BEGIN
   MachineConfig[0]."Unit Sep"."EM - 100"."L-GREEN".CW.ENABLE := True;
   MachineConfig[0]."Unit Sep"."EM - 100"."L-GREEN".CW.EXIST := False;
   MachineConfig[1].Machine."Family" := 1;
   MachineConfig[1].Machine.TypeNo := 1;
   MachineConfig[1].Machine.Range := 2;
   MachineConfig[1].Machine.SepType := 1;
   MachineConfig[1].Machine.Frame := 4;
   MachineConfig[1].Machine.DchSystem := 1;
   MachineConfig[1].Machine.Spare_1 := 1;
   MachineConfig[1].Machine.FeedPump := 1;
   MachineConfig[1].Machine.InlineCarbonation := 1;
   MachineConfig[1].Machine.eWON := 1;
   MachineConfig[1]."Unit Sep"."EM - 100"."L-GREEN".CW.ENABLE := true;
   MachineConfig[1]."Unit Sep"."EM - 100"."L-YELLOW".Tag := 'L-BLUE';
   MachineConfig[1]."Unit Sep"."EM - 100"."L-RED".CW.EXIST := True;
   MachineConfig[1]."Unit Sep"."EM - 100".EMS.CW.EXIST := True;
   MachineConfig[1]."Unit Sep"."EM - 100".EMS.Address := 180;
   MachineConfig[1]."Unit Sep"."EM - 100".UPS.CW.ENABLE := False;
   MachineConfig[1]."Unit Sep"."EM - 100".UPS.CW.EXIST := False;
   MachineConfig[1]."Unit Sep"."EM - 100".UPS.Address := 181;
   MachineConfig[1]."Unit Sep"."EM - 100".EWON.CW.ENABLE := True;
   MachineConfig[1]."Unit Sep"."EM - 100".EWON.CW.EXIST := True;
   MachineConfig[1]."Unit Sep"."EM - 100"."LT BUF".CW.ENABLE := False;
   MachineConfig[1]."Unit Sep"."EM - 400"."AV409-1".CW.ENABLE := False;
   MachineConfig[1]."Unit Sep"."EM - 400"."FCV409-1".CW.ENABLE := False;
   MachineConfig[1]."Unit Sep"."EM - 400"."FIS409-1".CW.ENABLE := false;
   MachineConfig[1]."Unit Sep"."EM - 400"."FIT409-1".CW.ENABLE := False;
   MachineConfig[1]."Unit Sep"."EM - 600"."AV615-1".ACT_OUT_ADD := 173;
   MachineConfig[1]."Unit Sep"."EM - 600"."AV63X/441-1".TAG := 'AV635-1';
   MachineConfig[1]."Unit Sep"."EM - 600"."AV63X/441-1".CW.ENABLE := True;
   MachineConfig[1]."Unit Sep"."EM - 600"."AV63X/441-1".ACT_OUT_ADD := 174;
   MachineConfig[1]."Unit Sep"."EM - 600"."FIS615-1".CW.ENABLE := false;
   MachineConfig[1]."Unit Sep"."EM - 600"."FIS635-1".CW.ENABLE := true;
   MachineConfig[1]."Unit Sep"."EM - 600"."FIS635-1".CW.EXIST := True;
   MachineConfig[1]."Unit Sep"."EM - 701".M701."TYPE" := 2;
   MachineConfig[1]."Unit Sep"."EM - 701".M701.FB_RUN_ADD := 8;
   MachineConfig[1]."Unit Sep"."EM - 701".M701.FB_RDY_ADD := 8;
   MachineConfig[1]."Unit Sep"."EM - 701".M701.OUT_ACT_ADD := 512;
   MachineConfig[1]."Unit Sep"."EM - 701".M701.OUT_RST_ADD := 8;
   MachineConfig[1]."Unit Sep"."EM - 701".M701_AMPS.CW.EXIST := True;
   MachineConfig[1]."Unit Sep"."EM - 730".TS730.CW.ENABLE := true;
   MachineConfig[1]."Unit Sep"."EM - 730".TS730.CW.EXIST := True;
   MachineConfig[1]."Unit Sep"."EM - 730".TS730.Address := 184;
   MachineConfig[1]."Unit Sep"."EM - 740"."P+F PS".Address := 180;
   MachineConfig[1]."Unit Sep"."EM - 740"."P+F OS".CW.EXIST := True;
   MachineConfig[1]."Unit Sep"."EM - 740"."P+F OS".Address := 182;
   MachineConfig[1]."Unit Sep"."EM - 740"."P+F ERROR".Address := 183;
   MachineConfig[1]."Unit Sep"."EM - 750".YT75X.CW.ENABLE := False;
   MachineConfig[1]."Unit Process"."EM - 201"."AV201-1".CW.ENABLE := true;
   MachineConfig[1]."Unit Process"."EM - 201"."AV201-1".CW.FB_CLS_EN := false;
   MachineConfig[1]."Unit Process"."EM - 201"."AV201-1".CW.FB_OPN_EN := false;
   MachineConfig[1]."Unit Process"."EM - 201"."AV201-1".CW.VLV_W_FB := false;
   MachineConfig[1]."Unit Process"."EM - 201"."AV201-1".FB_OPN_ADD := 8;
   MachineConfig[1]."Unit Process"."EM - 201"."AV201-1".FB_CLS_ADD := 8;
   MachineConfig[1]."Unit Process"."EM - 201"."AV201-1".ACT_OUT_ADD := 160;
   MachineConfig[1]."Unit Process"."EM - 201"."FCV201-1".CW.ENABLE := False;
   MachineConfig[1]."Unit Process"."EM - 201"."FIT201-1".CW.ENABLE := True;
   MachineConfig[1]."Unit Process"."EM - 201"."FIT201-1".CW.EXIST := True;
   MachineConfig[1]."Unit Process"."EM - 201"."FIT201-1"."Type" := 0;
   MachineConfig[1]."Unit Process"."EM - 201"."FIT201-1".Address := 88;
   MachineConfig[1]."Unit Process"."EM - 201"."FIT201-1".Max := 10000.0;
   MachineConfig[1]."Unit Process"."EM - 201"."LA201-1".CW.ENABLE := False;
   MachineConfig[1]."Unit Process"."EM - 201"."PIT201-1".CW.ENABLE := False;
   MachineConfig[1]."Unit Process"."EM - 22X"."FIT22X-1".CW.ENABLE := False;
   MachineConfig[1]."Unit Process"."EM - 22X"."PIT22X-1".CW.ENABLE := False;
   MachineConfig[1]."Unit Process"."EM - 22X"."QT220-1".CW.ENABLE := True;
   MachineConfig[1]."Unit Process"."EM - 22X"."QT220-1".CW.EXIST := False;
   MachineConfig[1]."Unit Process"."EM - 22X"."PCV22X-1".CW.ENABLE := False;
   MachineConfig[1]."Unit Process"."EM - 340"."AV340-1".CW.ENABLE := False;
   MachineConfig[1]."Unit Process"."EM - 340"."PIS340-1".Tag := 'PS301-1';
   MachineConfig[1]."Unit Process"."EM - 340"."PIS340-1".CW.INPUT := False;
   MachineConfig[1]."Unit Dch"."EM - 222"."LS222-1".CW.ENABLE := False;
   MachineConfig[1]."Unit Dch"."EM - 222"."P222-1".CW.EXIST := False;
   MachineConfig[1]."Unit Dch"."EM - 222"."P222-1".FB_RUN_ADD := 194;
   MachineConfig[1]."Unit Dch"."EM - 222"."P222-1".FB_RDY_ADD := 195;
   MachineConfig[1]."Unit Dch"."EM - 222"."P222-1".OUT_ACT_ADD := 182;
   MachineConfig[1]."Unit Dch"."EM - 222"."TS222-1".CW.ENABLE := False;
   MachineConfig[1]."Unit Dch"."EM - 222"."TT222-1".CW.ENABLE := False;
   MachineConfig[1]."Unit Dch"."EM - 300"."AV301-1".CW.ENABLE := True;
   MachineConfig[1]."Unit Dch"."EM - 300"."AV301-1".CW.FB_CLS_EN := false;
   MachineConfig[1]."Unit Dch"."EM - 300"."AV301-1".CW.FB_OPN_EN := false;
   MachineConfig[1]."Unit Dch"."EM - 300"."AV301-1".CW.VLV_W_FB := false;
   MachineConfig[1]."Unit Dch"."EM - 300"."AV301-1".FB_OPN_ADD := 8;
   MachineConfig[1]."Unit Dch"."EM - 300"."AV301-1".FB_CLS_ADD := 8;
   MachineConfig[1]."Unit Dch"."EM - 300"."AV301-1".ACT_OUT_ADD := 163;
   MachineConfig[1]."Unit Dch"."EM - 300"."AV304-1".ACT_OUT_ADD := 163;
   MachineConfig[1]."Unit Dch"."EM - 300"."AV320-1".CW.ENABLE := true;
   MachineConfig[1]."Unit Dch"."EM - 300"."AV320-1".CW.FB_CLS_EN := false;
   MachineConfig[1]."Unit Dch"."EM - 300"."AV320-1".CW.FB_OPN_EN := false;
   MachineConfig[1]."Unit Dch"."EM - 300"."AV320-1".CW.VLV_W_FB := false;
   MachineConfig[1]."Unit Dch"."EM - 300"."AV320-1".FB_OPN_ADD := 8;
   MachineConfig[1]."Unit Dch"."EM - 300"."AV320-1".FB_CLS_ADD := 8;
   MachineConfig[1]."Unit Dch"."EM - 300"."AV320-1".ACT_OUT_ADD := 164;
   MachineConfig[1]."Unit Dch"."EM - 300"."PS301-1".CW.ENABLE := True;
   MachineConfig[1]."Unit Dch"."EM - 300"."PS301-1".CW.EXIST := True;
   MachineConfig[1]."Unit Dch"."EM - 375"."AV37X-1".TAG := 'AV376-1';
   MachineConfig[1]."Unit Dch"."EM - 375"."AV37X-1".CW.ENABLE := true;
   MachineConfig[1]."Unit Dch"."EM - 375"."AV37X-1".ACT_OUT_ADD := 166;
   MachineConfig[1]."Unit Dch"."EM - 375".LS793.CW.ENABLE := True;
   MachineConfig[1]."Unit Dch"."EM - 375".LS793.CW.EXIST := True;
   MachineConfig[1]."Unit Dch"."EM - 375"."PIS375-1".CW.ENABLE := false;
   MachineConfig[1]."Unit Dch"."EM - 506".IP506a.CW.ENABLE := False;
   MachineConfig[1]."Unit Dch"."EM - 506".AVDCH.TAG := 'AV372-1';
   MachineConfig[1]."Unit Dch"."EM - 506".AVDCH.CW.ENABLE := True;
   MachineConfig[1]."Unit Dch"."EM - 506".AVDCH.ACT_OUT_ADD := 167;
   MachineConfig[1].Options."EM - P201"."P201-1".FB_RUN_ADD := 196;
   MachineConfig[1].Options."EM - P201"."P201-1".FB_RDY_ADD := 197;
   MachineConfig[1].Options."EM - P201"."P201-1".OUT_ACT_ADD := 183;
   MachineConfig[1].Options."EM - P201"."P201-1".OUT_RST_ADD := 184;
   MachineConfig[2].Machine."Family" := 1;
   MachineConfig[2].Machine.TypeNo := 2;
   MachineConfig[2].Machine.Range := 2;
   MachineConfig[2].Machine.SepType := 1;
   MachineConfig[2].Machine.Frame := 3;
   MachineConfig[2].Machine.DchSystem := 1;
   MachineConfig[2].Machine.Spare_1 := 1;
   MachineConfig[2].Machine.FeedPump := 1;
   MachineConfig[2].Machine.InlineCarbonation := 1;
   MachineConfig[2].Machine.eWON := 1;
   MachineConfig[2].Machine.ALBufferTank := 1;
   MachineConfig[2]."Unit Sep"."EM - 100"."L-GREEN".CW.ENABLE := true;
   MachineConfig[2]."Unit Sep"."EM - 100"."L-YELLOW".Tag := 'L-BLUE';
   MachineConfig[2]."Unit Sep"."EM - 100".EMS.Address := 180;
   MachineConfig[2]."Unit Sep"."EM - 100".UPS.CW.ENABLE := False;
   MachineConfig[2]."Unit Sep"."EM - 100".UPS.Address := 181;
   MachineConfig[2]."Unit Sep"."EM - 100".EWON.CW.ENABLE := True;
   MachineConfig[2]."Unit Sep"."EM - 100".EWON.CW.EXIST := True;
   MachineConfig[2]."Unit Sep"."EM - 400"."AV409-1".CW.ENABLE := False;
   MachineConfig[2]."Unit Sep"."EM - 400"."FCV409-1".CW.ENABLE := False;
   MachineConfig[2]."Unit Sep"."EM - 400"."FIS409-1".CW.ENABLE := false;
   MachineConfig[2]."Unit Sep"."EM - 400"."FIT409-1".CW.ENABLE := False;
   MachineConfig[2]."Unit Sep"."EM - 600"."AV63X/441-1".TAG := 'AV635-1';
   MachineConfig[2]."Unit Sep"."EM - 600"."AV63X/441-1".CW.ENABLE := True;
   MachineConfig[2]."Unit Sep"."EM - 600"."AV63X/441-1".ACT_OUT_ADD := 174;
   MachineConfig[2]."Unit Sep"."EM - 600"."FIS615-1".CW.ENABLE := False;
   MachineConfig[2]."Unit Sep"."EM - 600"."FIS635-1".CW.ENABLE := True;
   MachineConfig[2]."Unit Sep"."EM - 600"."FIS635-1".CW.EXIST := True;
   MachineConfig[2]."Unit Sep"."EM - 701".M701."TYPE" := 2;
   MachineConfig[2]."Unit Sep"."EM - 701".M701.FB_RUN_ADD := 8;
   MachineConfig[2]."Unit Sep"."EM - 701".M701.FB_RDY_ADD := 8;
   MachineConfig[2]."Unit Sep"."EM - 701".M701.OUT_ACT_ADD := 512;
   MachineConfig[2]."Unit Sep"."EM - 701".M701.OUT_RST_ADD := 8;
   MachineConfig[2]."Unit Sep"."EM - 730".TS730.CW.ENABLE := true;
   MachineConfig[2]."Unit Sep"."EM - 730".TS730.Address := 184;
   MachineConfig[2]."Unit Sep"."EM - 740"."P+F PS".Address := 180;
   MachineConfig[2]."Unit Sep"."EM - 740"."P+F OS".Address := 182;
   MachineConfig[2]."Unit Sep"."EM - 740"."P+F ERROR".Address := 183;
   MachineConfig[2]."Unit Sep"."EM - 750".YT75X.Tag := 'YT752';
   MachineConfig[2]."Unit Sep"."EM - 750".YT75X.CW.ENABLE := True;
   MachineConfig[2]."Unit Sep"."EM - 750".YT75X.Address := 78;
   MachineConfig[2]."Unit Sep"."EM - 750".YT75X.Min := 2.3;
   MachineConfig[2]."Unit Sep"."EM - 750".YT75X.Max := 5.5;
   MachineConfig[2]."Unit Sep"."EM - 750".YT75X.EU := 51;
   MachineConfig[2]."Unit Process"."EM - 201"."AV201-1".CW.ENABLE := True;
   MachineConfig[2]."Unit Process"."EM - 201"."AV201-1".CW.FB_CLS_EN := false;
   MachineConfig[2]."Unit Process"."EM - 201"."AV201-1".CW.FB_OPN_EN := false;
   MachineConfig[2]."Unit Process"."EM - 201"."AV201-1".CW.VLV_W_FB := false;
   MachineConfig[2]."Unit Process"."EM - 201"."AV201-1".FB_OPN_ADD := 8;
   MachineConfig[2]."Unit Process"."EM - 201"."AV201-1".FB_CLS_ADD := 8;
   MachineConfig[2]."Unit Process"."EM - 201"."AV201-1".ACT_OUT_ADD := 160;
   MachineConfig[2]."Unit Process"."EM - 201"."FCV201-1".CW.EXIST := false;
   MachineConfig[2]."Unit Process"."EM - 201"."FIT201-1"."Type" := 0;
   MachineConfig[2]."Unit Process"."EM - 201"."FIT201-1".Address := 88;
   MachineConfig[2]."Unit Process"."EM - 201"."FIT201-1".Max := 10000.0;
   MachineConfig[2]."Unit Process"."EM - 201"."LA201-1".CW.ENABLE := False;
   MachineConfig[2]."Unit Process"."EM - 201"."PIT201-1".CW.ENABLE := true;
   MachineConfig[2]."Unit Process"."EM - 201"."PIT201-1".CW.EXIST := false;
   MachineConfig[2]."Unit Process"."EM - 201"."QT201-1".CW.ENABLE := True;
   MachineConfig[2]."Unit Process"."EM - 22X"."AV220-1".CW.FB_CLS_EN := false;
   MachineConfig[2]."Unit Process"."EM - 22X"."AV220-1".CW.FB_OPN_EN := false;
   MachineConfig[2]."Unit Process"."EM - 22X"."AV220-1".CW.VLV_W_FB := false;
   MachineConfig[2]."Unit Process"."EM - 22X"."AV220-1".FB_OPN_ADD := 8;
   MachineConfig[2]."Unit Process"."EM - 22X"."AV220-1".FB_CLS_ADD := 8;
   MachineConfig[2]."Unit Process"."EM - 22X"."AV220-1".ACT_OUT_ADD := 162;
   MachineConfig[2]."Unit Process"."EM - 22X"."FIT22X-1".CW.ENABLE := false;
   MachineConfig[2]."Unit Process"."EM - 22X"."PIT22X-1".CW.EXIST := False;
   MachineConfig[2]."Unit Process"."EM - 22X"."QT220-1".CW.ENABLE := True;
   MachineConfig[2]."Unit Process"."EM - 22X"."QT220-1".CW.EXIST := False;
   MachineConfig[2]."Unit Process"."EM - 22X"."PCV22X-1".CW.ENABLE := False;
   MachineConfig[2]."Unit Process"."EM - 340"."AV340-1".CW.ENABLE := false;
   MachineConfig[2]."Unit Process"."EM - 340"."AV340-1".CW.FB_CLS_EN := false;
   MachineConfig[2]."Unit Process"."EM - 340"."AV340-1".CW.FB_OPN_EN := false;
   MachineConfig[2]."Unit Process"."EM - 340"."AV340-1".CW.EXIST := false;
   MachineConfig[2]."Unit Process"."EM - 340"."AV340-1".CW.VLV_W_FB := false;
   MachineConfig[2]."Unit Process"."EM - 340"."AV340-1".FB_OPN_ADD := 8;
   MachineConfig[2]."Unit Process"."EM - 340"."AV340-1".FB_CLS_ADD := 8;
   MachineConfig[2]."Unit Process"."EM - 340"."AV340-1".ACT_OUT_ADD := 8;
   MachineConfig[2]."Unit Dch"."EM - 222"."LS222-1".CW.ENABLE := False;
   MachineConfig[2]."Unit Dch"."EM - 222"."P222-1".CW.EXIST := False;
   MachineConfig[2]."Unit Dch"."EM - 222"."P222-1".FB_RUN_ADD := 194;
   MachineConfig[2]."Unit Dch"."EM - 222"."P222-1".FB_RDY_ADD := 195;
   MachineConfig[2]."Unit Dch"."EM - 222"."P222-1".OUT_ACT_ADD := 182;
   MachineConfig[2]."Unit Dch"."EM - 222"."TS222-1".CW.ENABLE := False;
   MachineConfig[2]."Unit Dch"."EM - 222"."TT222-1".CW.ENABLE := False;
   MachineConfig[2]."Unit Dch"."EM - 300"."AV301-1".TAG := 'AV301-1';
   MachineConfig[2]."Unit Dch"."EM - 300"."AV301-1".CW.ENABLE := True;
   MachineConfig[2]."Unit Dch"."EM - 300"."AV301-1".CW.FB_CLS_EN := false;
   MachineConfig[2]."Unit Dch"."EM - 300"."AV301-1".CW.FB_OPN_EN := false;
   MachineConfig[2]."Unit Dch"."EM - 300"."AV301-1".CW.VLV_W_FB := false;
   MachineConfig[2]."Unit Dch"."EM - 300"."AV301-1".FB_OPN_ADD := 8;
   MachineConfig[2]."Unit Dch"."EM - 300"."AV301-1".FB_CLS_ADD := 8;
   MachineConfig[2]."Unit Dch"."EM - 300"."AV301-1".ACT_OUT_ADD := 163;
   MachineConfig[2]."Unit Dch"."EM - 300"."AV304-1".ACT_OUT_ADD := 8;
   MachineConfig[2]."Unit Dch"."EM - 300"."AV320-1".CW.ENABLE := True;
   MachineConfig[2]."Unit Dch"."EM - 300"."AV320-1".CW.FB_CLS_EN := false;
   MachineConfig[2]."Unit Dch"."EM - 300"."AV320-1".CW.FB_OPN_EN := false;
   MachineConfig[2]."Unit Dch"."EM - 300"."AV320-1".CW.VLV_W_FB := false;
   MachineConfig[2]."Unit Dch"."EM - 300"."AV320-1".FB_OPN_ADD := 8;
   MachineConfig[2]."Unit Dch"."EM - 300"."AV320-1".FB_CLS_ADD := 8;
   MachineConfig[2]."Unit Dch"."EM - 300"."AV320-1".ACT_OUT_ADD := 164;
   MachineConfig[2]."Unit Dch"."EM - 300"."PS301-1".CW.ENABLE := True;
   MachineConfig[2]."Unit Dch"."EM - 300"."PS301-1".CW.EXIST := True;
   MachineConfig[2]."Unit Dch"."EM - 375"."AV37X-1".TAG := 'AV376-1';
   MachineConfig[2]."Unit Dch"."EM - 375"."AV37X-1".CW.ENABLE := true;
   MachineConfig[2]."Unit Dch"."EM - 375"."AV37X-1".ACT_OUT_ADD := 166;
   MachineConfig[2]."Unit Dch"."EM - 375"."PIS375-1".CW.ENABLE := false;
   MachineConfig[2]."Unit Dch"."EM - 506".IP506a.CW.ENABLE := False;
   MachineConfig[2]."Unit Dch"."EM - 506".AVDCH.TAG := 'AV372-1';
   MachineConfig[2]."Unit Dch"."EM - 506".AVDCH.CW.ENABLE := true;
   MachineConfig[2]."Unit Dch"."EM - 506".AVDCH.ACT_OUT_ADD := 167;
   MachineConfig[2].Options."EM - P201"."P201-1".FB_RUN_ADD := 196;
   MachineConfig[2].Options."EM - P201"."P201-1".FB_RDY_ADD := 197;
   MachineConfig[2].Options."EM - P201"."P201-1".OUT_ACT_ADD := 183;
   MachineConfig[2].Options."EM - P201"."P201-1".OUT_RST_ADD := 184;
   MachineConfig[2].Options."EM - 551"."FIT551-1".Address := 90;
   MachineConfig[2].Options."EM - 551"."FIT551-1".Max := 15000.0;
   MachineConfig[3]."Unit Sep"."EM - 100"."L-GREEN".CW.ENABLE := True;
   MachineConfig[3]."Unit Sep"."EM - 400"."FCV409-1".CW.ENABLE := false;
   MachineConfig[3]."Unit Sep"."EM - 730".TS730.CW.ENABLE := True;
   MachineConfig[3]."Unit Process"."EM - 201"."FIT201-1".Address := 88;
   MachineConfig[3]."Unit Process"."EM - 201"."FIT201-1".Max := 10000.0;
   MachineConfig[3]."Unit Dch"."EM - 222"."P222-1".CW.EXIST := false;
   MachineConfig[3]."Unit Dch"."EM - 300"."AV301-1".FB_OPN_ADD := 8;
   MachineConfig[3]."Unit Dch"."EM - 300"."AV301-1".FB_CLS_ADD := 8;
   MachineConfig[3]."Unit Dch"."EM - 300"."AV301-1".ACT_OUT_ADD := 163;
   MachineConfig[4].Machine."Family" := 1;
   MachineConfig[4].Machine.TypeNo := 4;
   MachineConfig[4].Machine.Range := 2;
   MachineConfig[4].Machine.SepType := 1;
   MachineConfig[4].Machine.Frame := 1;
   MachineConfig[4].Machine.DchSystem := 2;
   MachineConfig[4].Machine.Spare_1 := 1;
   MachineConfig[4].Machine.FeedPump := 1;
   MachineConfig[4].Machine.Spare_2 := 2;
   MachineConfig[4].Machine.InlineCarbonation := 1;
   MachineConfig[4].Machine.eWON := 1;
   MachineConfig[4].Machine.ALBufferTank := 1;
   MachineConfig[4]."Unit Sep"."EM - 100"."L-GREEN".CW.ENABLE := True;
   MachineConfig[4]."Unit Sep"."EM - 100"."L-YELLOW".Tag := 'L-BLUE';
   MachineConfig[4]."Unit Sep"."EM - 100".EMS.Address := 180;
   MachineConfig[4]."Unit Sep"."EM - 100".UPS.CW.ENABLE := True;
   MachineConfig[4]."Unit Sep"."EM - 100".UPS.CW.EXIST := True;
   MachineConfig[4]."Unit Sep"."EM - 100".UPS.Address := 181;
   MachineConfig[4]."Unit Sep"."EM - 100".EWON.CW.ENABLE := True;
   MachineConfig[4]."Unit Sep"."EM - 100".EWON.CW.EXIST := True;
   MachineConfig[4]."Unit Sep"."EM - 400"."AV409-1".CW.ENABLE := True;
   MachineConfig[4]."Unit Sep"."EM - 400"."AV409-1".ACT_OUT_ADD := 170;
   MachineConfig[4]."Unit Sep"."EM - 400"."FCV409-1".CW.ENABLE := True;
   MachineConfig[4]."Unit Sep"."EM - 400"."FCV409-1"."Type" := 0;
   MachineConfig[4]."Unit Sep"."EM - 400"."FCV409-1".Address := 78;
   MachineConfig[4]."Unit Sep"."EM - 400"."FCV409-1".Min := 0.0;
   MachineConfig[4]."Unit Sep"."EM - 400"."FCV409-1".Max := 100.0;
   MachineConfig[4]."Unit Sep"."EM - 400"."FIS409-1".CW.ENABLE := false;
   MachineConfig[4]."Unit Sep"."EM - 400"."FIT409-1".CW.ENABLE := True;
   MachineConfig[4]."Unit Sep"."EM - 400"."FIT409-1".CW.EXIST := True;
   MachineConfig[4]."Unit Sep"."EM - 400"."FIT409-1"."Type" := 0;
   MachineConfig[4]."Unit Sep"."EM - 400"."FIT409-1".Address := 92;
   MachineConfig[4]."Unit Sep"."EM - 400"."FIT409-1".Min := 24.0;
   MachineConfig[4]."Unit Sep"."EM - 400"."FIT409-1".Max := 252.0;
   MachineConfig[4]."Unit Sep"."EM - 400"."TT41X-1".CW.ENABLE := True;
   MachineConfig[4]."Unit Sep"."EM - 400"."TT41X-1"."Type" := 0;
   MachineConfig[4]."Unit Sep"."EM - 400"."TT41X-1".Address := 86;
   MachineConfig[4]."Unit Sep"."EM - 400"."TT41X-1".Min := -50.0;
   MachineConfig[4]."Unit Sep"."EM - 400"."TT41X-1".Max := 150.0;
   MachineConfig[4]."Unit Sep"."EM - 600"."AV615-1".CW.ENABLE := True;
   MachineConfig[4]."Unit Sep"."EM - 600"."AV615-1".ACT_OUT_ADD := 173;
   MachineConfig[4]."Unit Sep"."EM - 600"."AV63X/441-1".TAG := 'AV635-1';
   MachineConfig[4]."Unit Sep"."EM - 600"."AV63X/441-1".CW.ENABLE := true;
   MachineConfig[4]."Unit Sep"."EM - 600"."AV63X/441-1".ACT_OUT_ADD := 174;
   MachineConfig[4]."Unit Sep"."EM - 600"."FIS615-1".Tag := 'FS615-1';
   MachineConfig[4]."Unit Sep"."EM - 600"."FIS615-1".CW.ENABLE := True;
   MachineConfig[4]."Unit Sep"."EM - 600"."FIS635-1".Tag := 'FS635-1';
   MachineConfig[4]."Unit Sep"."EM - 600"."FIS635-1".CW.ENABLE := True;
   MachineConfig[4]."Unit Sep"."EM - 701".M701."TYPE" := 2;
   MachineConfig[4]."Unit Sep"."EM - 701".M701.FB_RUN_ADD := 8;
   MachineConfig[4]."Unit Sep"."EM - 701".M701.FB_RDY_ADD := 8;
   MachineConfig[4]."Unit Sep"."EM - 701".M701.OUT_ACT_ADD := 512;
   MachineConfig[4]."Unit Sep"."EM - 701".M701.OUT_RST_ADD := 8;
   MachineConfig[4]."Unit Sep"."EM - 730".TS730.CW.ENABLE := True;
   MachineConfig[4]."Unit Sep"."EM - 730".TS730.CW.EXIST := True;
   MachineConfig[4]."Unit Sep"."EM - 730".TS730.Address := 184;
   MachineConfig[4]."Unit Sep"."EM - 740"."P+F PS".Address := 180;
   MachineConfig[4]."Unit Sep"."EM - 740"."P+F OS".Address := 182;
   MachineConfig[4]."Unit Sep"."EM - 740"."P+F ERROR".Address := 183;
   MachineConfig[4]."Unit Sep"."EM - 750".YT75X.CW.ENABLE := True;
   MachineConfig[4]."Unit Sep"."EM - 750".YT75X.Address := 78;
   MachineConfig[4]."Unit Process"."EM - 201"."AV201-1".CW.ENABLE := True;
   MachineConfig[4]."Unit Process"."EM - 201"."AV201-1".CW.FB_CLS_EN := False;
   MachineConfig[4]."Unit Process"."EM - 201"."AV201-1".CW.FB_OPN_EN := False;
   MachineConfig[4]."Unit Process"."EM - 201"."AV201-1".CW.VLV_W_FB := False;
   MachineConfig[4]."Unit Process"."EM - 201"."AV201-1".FB_OPN_ADD := 8;
   MachineConfig[4]."Unit Process"."EM - 201"."AV201-1".FB_CLS_ADD := 8;
   MachineConfig[4]."Unit Process"."EM - 201"."AV201-1".ACT_OUT_ADD := 160;
   MachineConfig[4]."Unit Process"."EM - 201"."AV460a-1".CW.ENABLE := True;
   MachineConfig[4]."Unit Process"."EM - 201"."FCV201-1".CW.EXIST := False;
   MachineConfig[4]."Unit Process"."EM - 201"."FIT201-1"."Type" := 0;
   MachineConfig[4]."Unit Process"."EM - 201"."FIT201-1".Address := 88;
   MachineConfig[4]."Unit Process"."EM - 201"."FIT201-1".Max := 50000.0;
   MachineConfig[4]."Unit Process"."EM - 201"."LA201-1".CW.ENABLE := False;
   MachineConfig[4]."Unit Process"."EM - 201"."PIT201-1".CW.EXIST := false;
   MachineConfig[4]."Unit Process"."EM - 201"."QT201-1".CW.ENABLE := True;
   MachineConfig[4]."Unit Process"."EM - 212"."AV212-1".CW.ENABLE := True;
   MachineConfig[4]."Unit Process"."EM - 212"."AV212-1".CW.FB_CLS_EN := False;
   MachineConfig[4]."Unit Process"."EM - 212"."AV212-1".CW.FB_OPN_EN := False;
   MachineConfig[4]."Unit Process"."EM - 212"."AV212-1".CW.EXIST := False;
   MachineConfig[4]."Unit Process"."EM - 212"."AV212-1".CW.VLV_W_FB := False;
   MachineConfig[4]."Unit Process"."EM - 212"."AV212-1".FB_OPN_ADD := 8;
   MachineConfig[4]."Unit Process"."EM - 212"."AV212-1".FB_CLS_ADD := 8;
   MachineConfig[4]."Unit Process"."EM - 212"."AV212-1".ACT_OUT_ADD := 161;
   MachineConfig[4]."Unit Process"."EM - 22X"."AV220-1".CW.ENABLE := True;
   MachineConfig[4]."Unit Process"."EM - 22X"."AV220-1".CW.FB_CLS_EN := false;
   MachineConfig[4]."Unit Process"."EM - 22X"."AV220-1".CW.FB_OPN_EN := false;
   MachineConfig[4]."Unit Process"."EM - 22X"."AV220-1".CW.EXIST := false;
   MachineConfig[4]."Unit Process"."EM - 22X"."AV220-1".CW.VLV_W_FB := false;
   MachineConfig[4]."Unit Process"."EM - 22X"."AV220-1".FB_OPN_ADD := 8;
   MachineConfig[4]."Unit Process"."EM - 22X"."AV220-1".FB_CLS_ADD := 8;
   MachineConfig[4]."Unit Process"."EM - 22X"."AV220-1".ACT_OUT_ADD := 162;
   MachineConfig[4]."Unit Process"."EM - 22X"."AV460-1".CW.ENABLE := True;
   MachineConfig[4]."Unit Process"."EM - 22X"."AV460-1".CW.FB_CLS_EN := false;
   MachineConfig[4]."Unit Process"."EM - 22X"."AV460-1".CW.FB_OPN_EN := false;
   MachineConfig[4]."Unit Process"."EM - 22X"."AV460-1".CW.EXIST := false;
   MachineConfig[4]."Unit Process"."EM - 22X"."AV460-1".CW.VLV_W_FB := false;
   MachineConfig[4]."Unit Process"."EM - 22X"."AV460-1".FB_OPN_ADD := 8;
   MachineConfig[4]."Unit Process"."EM - 22X"."AV460-1".FB_CLS_ADD := 8;
   MachineConfig[4]."Unit Process"."EM - 22X"."AV460-1".ACT_OUT_ADD := 171;
   MachineConfig[4]."Unit Process"."EM - 22X"."FIT22X-1".CW.ENABLE := False;
   MachineConfig[4]."Unit Process"."EM - 22X"."PIT22X-1".CW.EXIST := false;
   MachineConfig[4]."Unit Process"."EM - 22X"."QT220-1".CW.ENABLE := True;
   MachineConfig[4]."Unit Process"."EM - 22X"."QT220-1".CW.EXIST := False;
   MachineConfig[4]."Unit Process"."EM - 22X"."PCV22X-1".CW.ENABLE := False;
   MachineConfig[4]."Unit Process"."EM - 340"."AV340-1".CW.ENABLE := True;
   MachineConfig[4]."Unit Process"."EM - 340"."AV340-1".CW.FB_CLS_EN := False;
   MachineConfig[4]."Unit Process"."EM - 340"."AV340-1".CW.FB_OPN_EN := False;
   MachineConfig[4]."Unit Process"."EM - 340"."AV340-1".CW.EXIST := False;
   MachineConfig[4]."Unit Process"."EM - 340"."AV340-1".CW.VLV_W_FB := False;
   MachineConfig[4]."Unit Process"."EM - 340"."AV340-1".FB_OPN_ADD := 8;
   MachineConfig[4]."Unit Process"."EM - 340"."AV340-1".FB_CLS_ADD := 8;
   MachineConfig[4]."Unit Process"."EM - 340"."AV340-1".ACT_OUT_ADD := 165;
   MachineConfig[4]."Unit Process"."EM - 340"."PIS340-1".Tag := 'PS301-1';
   MachineConfig[4]."Unit Dch"."EM - 222"."LS222-1".CW.ENABLE := False;
   MachineConfig[4]."Unit Dch"."EM - 222"."P222-1".CW.EXIST := False;
   MachineConfig[4]."Unit Dch"."EM - 222"."P222-1".FB_RUN_ADD := 194;
   MachineConfig[4]."Unit Dch"."EM - 222"."P222-1".FB_RDY_ADD := 195;
   MachineConfig[4]."Unit Dch"."EM - 222"."P222-1".OUT_ACT_ADD := 182;
   MachineConfig[4]."Unit Dch"."EM - 222"."TS222-1".CW.ENABLE := False;
   MachineConfig[4]."Unit Dch"."EM - 222"."TT222-1".CW.ENABLE := False;
   MachineConfig[4]."Unit Dch"."EM - 300"."AV301-1".CW.ENABLE := True;
   MachineConfig[4]."Unit Dch"."EM - 300"."AV301-1".CW.FB_CLS_EN := False;
   MachineConfig[4]."Unit Dch"."EM - 300"."AV301-1".CW.FB_OPN_EN := False;
   MachineConfig[4]."Unit Dch"."EM - 300"."AV301-1".CW.VLV_W_FB := False;
   MachineConfig[4]."Unit Dch"."EM - 300"."AV301-1".FB_OPN_ADD := 8;
   MachineConfig[4]."Unit Dch"."EM - 300"."AV301-1".FB_CLS_ADD := 8;
   MachineConfig[4]."Unit Dch"."EM - 300"."AV301-1".ACT_OUT_ADD := 163;
   MachineConfig[4]."Unit Dch"."EM - 300"."AV304-1".TAG := 'AV301-1';
   MachineConfig[4]."Unit Dch"."EM - 300"."AV304-1".ACT_OUT_ADD := 163;
   MachineConfig[4]."Unit Dch"."EM - 300"."AV320-1".CW.ENABLE := True;
   MachineConfig[4]."Unit Dch"."EM - 300"."AV320-1".CW.FB_CLS_EN := false;
   MachineConfig[4]."Unit Dch"."EM - 300"."AV320-1".CW.FB_OPN_EN := false;
   MachineConfig[4]."Unit Dch"."EM - 300"."AV320-1".CW.VLV_W_FB := false;
   MachineConfig[4]."Unit Dch"."EM - 300"."AV320-1".FB_OPN_ADD := 8;
   MachineConfig[4]."Unit Dch"."EM - 300"."AV320-1".FB_CLS_ADD := 8;
   MachineConfig[4]."Unit Dch"."EM - 300"."AV320-1".ACT_OUT_ADD := 164;
   MachineConfig[4]."Unit Dch"."EM - 300"."AV635-1".ACT_OUT_ADD := 174;
   MachineConfig[4]."Unit Dch"."EM - 375"."AV37X-1".TAG := 'AV375-1';
   MachineConfig[4]."Unit Dch"."EM - 375"."AV37X-1".CW.ENABLE := true;
   MachineConfig[4]."Unit Dch"."EM - 375"."AV37X-1".ACT_OUT_ADD := 166;
   MachineConfig[4]."Unit Dch"."EM - 375"."PIS375-1".CW.ENABLE := false;
   MachineConfig[4]."Unit Dch"."EM - 375"."PT37X-1".Tag := 'PT375-1';
   MachineConfig[4]."Unit Dch"."EM - 375"."PT37X-1".CW.ENABLE := True;
   MachineConfig[4]."Unit Dch"."EM - 375"."PT37X-1".CW.EXIST := True;
   MachineConfig[4]."Unit Dch"."EM - 375"."PT37X-1".Address := 76;
   MachineConfig[4]."Unit Dch"."EM - 375"."PT37X-1".Max := 600.0;
   MachineConfig[4]."Unit Dch"."EM - 506".IP506a.CW.ENABLE := True;
   MachineConfig[4]."Unit Dch"."EM - 506".IP506a.CW.EXIST := True;
   MachineConfig[4]."Unit Dch"."EM - 506".AVDCH.TAG := '506b';
   MachineConfig[4]."Unit Dch"."EM - 506".AVDCH.CW.ENABLE := true;
   MachineConfig[4]."Unit Dch"."EM - 506".AVDCH.ACT_OUT_ADD := 167;
   MachineConfig[4].Options."EM - P201"."P201-1".FB_RUN_ADD := 196;
   MachineConfig[4].Options."EM - P201"."P201-1".FB_RDY_ADD := 197;
   MachineConfig[4].Options."EM - P201"."P201-1".OUT_ACT_ADD := 183;
   MachineConfig[4].Options."EM - P201"."P201-1".OUT_RST_ADD := 184;
   MachineConfig[5].Machine."Family" := 1;
   MachineConfig[5].Machine.TypeNo := 5;
   MachineConfig[5].Machine.Range := 2;
   MachineConfig[5].Machine.SepType := 1;
   MachineConfig[5].Machine.Frame := 1;
   MachineConfig[5].Machine.DchSystem := 2;
   MachineConfig[5].Machine.Spare_1 := 1;
   MachineConfig[5].Machine.FeedPump := 1;
   MachineConfig[5].Machine.Spare_2 := 2;
   MachineConfig[5].Machine.InlineCarbonation := 1;
   MachineConfig[5].Machine.eWON := 1;
   MachineConfig[5].Machine.ALBufferTank := 1;
   MachineConfig[5]."Unit Sep"."EM - 100"."L-GREEN".CW.ENABLE := True;
   MachineConfig[5]."Unit Sep"."EM - 100"."L-GREEN".CW.EXIST := True;
   MachineConfig[5]."Unit Sep"."EM - 100"."L-YELLOW".Tag := 'L-BLUE';
   MachineConfig[5]."Unit Sep"."EM - 100".EMS.Address := 180;
   MachineConfig[5]."Unit Sep"."EM - 100".UPS.CW.ENABLE := True;
   MachineConfig[5]."Unit Sep"."EM - 100".UPS.CW.EXIST := True;
   MachineConfig[5]."Unit Sep"."EM - 100".UPS.Address := 181;
   MachineConfig[5]."Unit Sep"."EM - 100".EWON.CW.ENABLE := True;
   MachineConfig[5]."Unit Sep"."EM - 100".EWON.CW.EXIST := True;
   MachineConfig[5]."Unit Sep"."EM - 400"."AV409-1".CW.ENABLE := True;
   MachineConfig[5]."Unit Sep"."EM - 400"."AV409-1".ACT_OUT_ADD := 170;
   MachineConfig[5]."Unit Sep"."EM - 400"."FCV409-1".CW.ENABLE := True;
   MachineConfig[5]."Unit Sep"."EM - 400"."FCV409-1".CW.EXIST := True;
   MachineConfig[5]."Unit Sep"."EM - 400"."FCV409-1"."Type" := 0;
   MachineConfig[5]."Unit Sep"."EM - 400"."FCV409-1".Address := 78;
   MachineConfig[5]."Unit Sep"."EM - 400"."FCV409-1".Min := 0.0;
   MachineConfig[5]."Unit Sep"."EM - 400"."FCV409-1".Max := 100.0;
   MachineConfig[5]."Unit Sep"."EM - 400"."FIS409-1".CW.ENABLE := false;
   MachineConfig[5]."Unit Sep"."EM - 400"."FIT409-1".CW.ENABLE := True;
   MachineConfig[5]."Unit Sep"."EM - 400"."FIT409-1".CW.EXIST := True;
   MachineConfig[5]."Unit Sep"."EM - 400"."FIT409-1"."Type" := 0;
   MachineConfig[5]."Unit Sep"."EM - 400"."FIT409-1".Address := 92;
   MachineConfig[5]."Unit Sep"."EM - 400"."FIT409-1".Min := 24.0;
   MachineConfig[5]."Unit Sep"."EM - 400"."FIT409-1".Max := 252.0;
   MachineConfig[5]."Unit Sep"."EM - 400"."TT41X-1".CW.ENABLE := True;
   MachineConfig[5]."Unit Sep"."EM - 400"."TT41X-1"."Type" := 0;
   MachineConfig[5]."Unit Sep"."EM - 400"."TT41X-1".Address := 86;
   MachineConfig[5]."Unit Sep"."EM - 400"."TT41X-1".Min := -50.0;
   MachineConfig[5]."Unit Sep"."EM - 400"."TT41X-1".Max := 150.0;
   MachineConfig[5]."Unit Sep"."EM - 600"."AV615-1".CW.ENABLE := True;
   MachineConfig[5]."Unit Sep"."EM - 600"."AV615-1".ACT_OUT_ADD := 173;
   MachineConfig[5]."Unit Sep"."EM - 600"."AV63X/441-1".TAG := 'AV635-1';
   MachineConfig[5]."Unit Sep"."EM - 600"."AV63X/441-1".CW.ENABLE := true;
   MachineConfig[5]."Unit Sep"."EM - 600"."AV63X/441-1".ACT_OUT_ADD := 174;
   MachineConfig[5]."Unit Sep"."EM - 600"."FIS615-1".Tag := 'FS615-1';
   MachineConfig[5]."Unit Sep"."EM - 600"."FIS615-1".CW.ENABLE := True;
   MachineConfig[5]."Unit Sep"."EM - 600"."FIS635-1".Tag := 'FS635-1';
   MachineConfig[5]."Unit Sep"."EM - 600"."FIS635-1".CW.ENABLE := True;
   MachineConfig[5]."Unit Sep"."EM - 701".M701."TYPE" := 2;
   MachineConfig[5]."Unit Sep"."EM - 701".M701.FB_RUN_ADD := 8;
   MachineConfig[5]."Unit Sep"."EM - 701".M701.FB_RDY_ADD := 8;
   MachineConfig[5]."Unit Sep"."EM - 701".M701.OUT_ACT_ADD := 512;
   MachineConfig[5]."Unit Sep"."EM - 701".M701.OUT_RST_ADD := 8;
   MachineConfig[5]."Unit Sep"."EM - 730".TS730.CW.ENABLE := True;
   MachineConfig[5]."Unit Sep"."EM - 730".TS730.CW.EXIST := True;
   MachineConfig[5]."Unit Sep"."EM - 730".TS730.Address := 184;
   MachineConfig[5]."Unit Sep"."EM - 740"."P+F PS".Address := 180;
   MachineConfig[5]."Unit Sep"."EM - 740"."P+F OS".Address := 182;
   MachineConfig[5]."Unit Sep"."EM - 740"."P+F ERROR".Address := 183;
   MachineConfig[5]."Unit Sep"."EM - 750".YT75X.CW.ENABLE := True;
   MachineConfig[5]."Unit Sep"."EM - 750".YT75X.Address := 78;
   MachineConfig[5]."Unit Process"."EM - 201"."AV201-1".CW.ENABLE := True;
   MachineConfig[5]."Unit Process"."EM - 201"."AV201-1".CW.FB_CLS_EN := False;
   MachineConfig[5]."Unit Process"."EM - 201"."AV201-1".CW.FB_OPN_EN := False;
   MachineConfig[5]."Unit Process"."EM - 201"."AV201-1".CW.VLV_W_FB := False;
   MachineConfig[5]."Unit Process"."EM - 201"."AV201-1".FB_OPN_ADD := 8;
   MachineConfig[5]."Unit Process"."EM - 201"."AV201-1".FB_CLS_ADD := 8;
   MachineConfig[5]."Unit Process"."EM - 201"."AV201-1".ACT_OUT_ADD := 160;
   MachineConfig[5]."Unit Process"."EM - 201"."AV460a-1".CW.ENABLE := True;
   MachineConfig[5]."Unit Process"."EM - 201"."FIT201-1"."Type" := 0;
   MachineConfig[5]."Unit Process"."EM - 201"."FIT201-1".Address := 88;
   MachineConfig[5]."Unit Process"."EM - 201"."FIT201-1".Max := 50000.0;
   MachineConfig[5]."Unit Process"."EM - 201"."LA201-1".CW.ENABLE := False;
   MachineConfig[5]."Unit Process"."EM - 201"."QT201-1".CW.ENABLE := True;
   MachineConfig[5]."Unit Process"."EM - 201"."QT201-1".CW.EXIST := True;
   MachineConfig[5]."Unit Process"."EM - 212"."AV212-1".CW.ENABLE := True;
   MachineConfig[5]."Unit Process"."EM - 212"."AV212-1".CW.FB_CLS_EN := False;
   MachineConfig[5]."Unit Process"."EM - 212"."AV212-1".CW.FB_OPN_EN := False;
   MachineConfig[5]."Unit Process"."EM - 212"."AV212-1".CW.EXIST := False;
   MachineConfig[5]."Unit Process"."EM - 212"."AV212-1".CW.VLV_W_FB := False;
   MachineConfig[5]."Unit Process"."EM - 212"."AV212-1".FB_OPN_ADD := 8;
   MachineConfig[5]."Unit Process"."EM - 212"."AV212-1".FB_CLS_ADD := 8;
   MachineConfig[5]."Unit Process"."EM - 212"."AV212-1".ACT_OUT_ADD := 161;
   MachineConfig[5]."Unit Process"."EM - 22X"."AV220-1".CW.ENABLE := True;
   MachineConfig[5]."Unit Process"."EM - 22X"."AV220-1".CW.FB_CLS_EN := false;
   MachineConfig[5]."Unit Process"."EM - 22X"."AV220-1".CW.FB_OPN_EN := false;
   MachineConfig[5]."Unit Process"."EM - 22X"."AV220-1".CW.VLV_W_FB := false;
   MachineConfig[5]."Unit Process"."EM - 22X"."AV220-1".FB_OPN_ADD := 8;
   MachineConfig[5]."Unit Process"."EM - 22X"."AV220-1".FB_CLS_ADD := 8;
   MachineConfig[5]."Unit Process"."EM - 22X"."AV220-1".ACT_OUT_ADD := 162;
   MachineConfig[5]."Unit Process"."EM - 22X"."AV460-1".CW.ENABLE := True;
   MachineConfig[5]."Unit Process"."EM - 22X"."AV460-1".CW.FB_CLS_EN := false;
   MachineConfig[5]."Unit Process"."EM - 22X"."AV460-1".CW.FB_OPN_EN := false;
   MachineConfig[5]."Unit Process"."EM - 22X"."AV460-1".CW.VLV_W_FB := false;
   MachineConfig[5]."Unit Process"."EM - 22X"."AV460-1".FB_OPN_ADD := 8;
   MachineConfig[5]."Unit Process"."EM - 22X"."AV460-1".FB_CLS_ADD := 8;
   MachineConfig[5]."Unit Process"."EM - 22X"."AV460-1".ACT_OUT_ADD := 171;
   MachineConfig[5]."Unit Process"."EM - 22X"."FIT22X-1".CW.ENABLE := false;
   MachineConfig[5]."Unit Process"."EM - 22X"."PIT22X-1".Tag := 'PIT220-1';
   MachineConfig[5]."Unit Process"."EM - 22X"."PIT22X-1".CW.ENABLE := True;
   MachineConfig[5]."Unit Process"."EM - 22X"."PIT22X-1".Address := 66;
   MachineConfig[5]."Unit Process"."EM - 22X"."QT220-1".Tag := 'QT220-1';
   MachineConfig[5]."Unit Process"."EM - 22X"."QT220-1".CW.ENABLE := True;
   MachineConfig[5]."Unit Process"."EM - 22X"."QT220-1".Address := 70;
   MachineConfig[5]."Unit Process"."EM - 22X"."PCV22X-1".CW.ENABLE := False;
   MachineConfig[5]."Unit Process"."EM - 340"."AV340-1".CW.ENABLE := True;
   MachineConfig[5]."Unit Process"."EM - 340"."AV340-1".CW.FB_CLS_EN := False;
   MachineConfig[5]."Unit Process"."EM - 340"."AV340-1".CW.FB_OPN_EN := False;
   MachineConfig[5]."Unit Process"."EM - 340"."AV340-1".CW.VLV_W_FB := False;
   MachineConfig[5]."Unit Process"."EM - 340"."AV340-1".FB_OPN_ADD := 8;
   MachineConfig[5]."Unit Process"."EM - 340"."AV340-1".FB_CLS_ADD := 8;
   MachineConfig[5]."Unit Process"."EM - 340"."AV340-1".ACT_OUT_ADD := 165;
   MachineConfig[5]."Unit Process"."EM - 340"."PIS340-1".Tag := 'PS301-1';
   MachineConfig[5]."Unit Dch"."EM - 222"."LS222-1".CW.ENABLE := False;
   MachineConfig[5]."Unit Dch"."EM - 222"."P222-1".FB_RUN_ADD := 194;
   MachineConfig[5]."Unit Dch"."EM - 222"."P222-1".FB_RDY_ADD := 195;
   MachineConfig[5]."Unit Dch"."EM - 222"."P222-1".OUT_ACT_ADD := 182;
   MachineConfig[5]."Unit Dch"."EM - 222"."PIT222-1".CW.ENABLE := True;
   MachineConfig[5]."Unit Dch"."EM - 222"."TS222-1".CW.ENABLE := False;
   MachineConfig[5]."Unit Dch"."EM - 222"."TT222-1".CW.ENABLE := True;
   MachineConfig[5]."Unit Dch"."EM - 300"."AV301-1".CW.ENABLE := True;
   MachineConfig[5]."Unit Dch"."EM - 300"."AV301-1".CW.FB_CLS_EN := False;
   MachineConfig[5]."Unit Dch"."EM - 300"."AV301-1".CW.FB_OPN_EN := False;
   MachineConfig[5]."Unit Dch"."EM - 300"."AV301-1".CW.VLV_W_FB := False;
   MachineConfig[5]."Unit Dch"."EM - 300"."AV301-1".FB_OPN_ADD := 8;
   MachineConfig[5]."Unit Dch"."EM - 300"."AV301-1".FB_CLS_ADD := 8;
   MachineConfig[5]."Unit Dch"."EM - 300"."AV301-1".ACT_OUT_ADD := 163;
   MachineConfig[5]."Unit Dch"."EM - 300"."AV304-1".TAG := 'AV301-1';
   MachineConfig[5]."Unit Dch"."EM - 300"."AV304-1".ACT_OUT_ADD := 163;
   MachineConfig[5]."Unit Dch"."EM - 300"."AV320-1".CW.ENABLE := true;
   MachineConfig[5]."Unit Dch"."EM - 300"."AV320-1".CW.FB_CLS_EN := false;
   MachineConfig[5]."Unit Dch"."EM - 300"."AV320-1".CW.FB_OPN_EN := false;
   MachineConfig[5]."Unit Dch"."EM - 300"."AV320-1".CW.VLV_W_FB := false;
   MachineConfig[5]."Unit Dch"."EM - 300"."AV320-1".FB_OPN_ADD := 8;
   MachineConfig[5]."Unit Dch"."EM - 300"."AV320-1".FB_CLS_ADD := 8;
   MachineConfig[5]."Unit Dch"."EM - 300"."AV320-1".ACT_OUT_ADD := 164;
   MachineConfig[5]."Unit Dch"."EM - 300"."AV635-1".ACT_OUT_ADD := 174;
   MachineConfig[5]."Unit Dch"."EM - 375"."AV37X-1".TAG := 'AV375-1';
   MachineConfig[5]."Unit Dch"."EM - 375"."AV37X-1".CW.ENABLE := true;
   MachineConfig[5]."Unit Dch"."EM - 375"."AV37X-1".ACT_OUT_ADD := 166;
   MachineConfig[5]."Unit Dch"."EM - 375"."PIS375-1".CW.ENABLE := false;
   MachineConfig[5]."Unit Dch"."EM - 375"."PT37X-1".Tag := 'PT375-1';
   MachineConfig[5]."Unit Dch"."EM - 375"."PT37X-1".CW.ENABLE := True;
   MachineConfig[5]."Unit Dch"."EM - 375"."PT37X-1".CW.EXIST := True;
   MachineConfig[5]."Unit Dch"."EM - 375"."PT37X-1".Address := 76;
   MachineConfig[5]."Unit Dch"."EM - 375"."PT37X-1".Max := 600.0;
   MachineConfig[5]."Unit Dch"."EM - 506".IP506a.CW.ENABLE := True;
   MachineConfig[5]."Unit Dch"."EM - 506".AVDCH.TAG := '506b';
   MachineConfig[5]."Unit Dch"."EM - 506".AVDCH.CW.ENABLE := true;
   MachineConfig[5]."Unit Dch"."EM - 506".AVDCH.ACT_OUT_ADD := 167;
   MachineConfig[5].Options."EM - P201"."P201-1".FB_RUN_ADD := 196;
   MachineConfig[5].Options."EM - P201"."P201-1".FB_RDY_ADD := 197;
   MachineConfig[5].Options."EM - P201"."P201-1".OUT_ACT_ADD := 183;
   MachineConfig[5].Options."EM - P201"."P201-1".OUT_RST_ADD := 184;
   MachineConfig[7].Machine."Family" := 1;
   MachineConfig[7].Machine.TypeNo := 7;
   MachineConfig[7].Machine.Range := 1;
   MachineConfig[7].Machine.SepType := 1;
   MachineConfig[7].Machine.Frame := 1;
   MachineConfig[7].Machine.DchSystem := 2;
   MachineConfig[7].Machine.Spare_1 := 1;
   MachineConfig[7].Machine.FeedPump := 1;
   MachineConfig[7].Machine.Blending := 1;
   MachineConfig[7].Machine.Recirculation := 1;
   MachineConfig[7].Machine.CoolingRecirculation := 1;
   MachineConfig[7].Machine.Spare_2 := 2;
   MachineConfig[7].Machine.ConditionAlert := 1;
   MachineConfig[7].Machine.eWON := 1;
   MachineConfig[7].Machine.ALBufferTank := 1;
   MachineConfig[7]."Unit Sep"."EM - 100"."L-GREEN".CW.ENABLE := True;
   MachineConfig[7]."Unit Sep"."EM - 100"."L-YELLOW".CW.ENABLE := True;
   MachineConfig[7]."Unit Sep"."EM - 100".UPS.CW.EXIST := True;
   MachineConfig[7]."Unit Sep"."EM - 400"."AV409-1".CW.ENABLE := true;
   MachineConfig[7]."Unit Sep"."EM - 400"."FCV409-1".CW.ENABLE := True;
   MachineConfig[7]."Unit Sep"."EM - 400"."FCV409-1".CW.EXIST := True;
   MachineConfig[7]."Unit Sep"."EM - 400"."FIT409-1".CW.ENABLE := True;
   MachineConfig[7]."Unit Sep"."EM - 400"."FIT409-1".CW.EXIST := True;
   MachineConfig[7]."Unit Sep"."EM - 400"."TT41X-1".CW.ENABLE := True;
   MachineConfig[7]."Unit Sep"."EM - 400"."TT41X-1".CW.EXIST := True;
   MachineConfig[7]."Unit Sep"."EM - 400"."TT41X-1".Address := 142;
   MachineConfig[7]."Unit Sep"."EM - 600"."AV615-1".CW.ENABLE := True;
   MachineConfig[7]."Unit Sep"."EM - 600"."FIS615-1".CW.ENABLE := True;
   MachineConfig[7]."Unit Sep"."EM - 600"."FIS635-1".CW.ENABLE := true;
   MachineConfig[7]."Unit Sep"."EM - 600"."FIS635-1".CW.EXIST := true;
   MachineConfig[7]."Unit Sep"."EM - 701".M701."TYPE" := 1;
   MachineConfig[7]."Unit Sep"."EM - 730".TS730.CW.ENABLE := True;
   MachineConfig[7]."Unit Sep"."EM - 730".TS730.CW.EXIST := True;
   MachineConfig[7]."Unit Sep"."EM - 750".YT75X.CW.ENABLE := True;
   MachineConfig[7]."Unit Process"."EM - 201"."AV201-1".CW.ENABLE := true;
   MachineConfig[7]."Unit Process"."EM - 201"."FIT201-1"."Type" := 2;
   MachineConfig[7]."Unit Process"."EM - 201"."FIT201-1".Address := 256;
   MachineConfig[7]."Unit Process"."EM - 201"."FIT201-1".Max := 65000.0;
   MachineConfig[7]."Unit Process"."EM - 201"."LA201-1".CW.ENABLE := true;
   MachineConfig[7]."Unit Process"."EM - 201"."QT201-1".CW.ENABLE := True;
   MachineConfig[7]."Unit Process"."EM - 201"."QT201-1".CW.EXIST := True;
   MachineConfig[7]."Unit Process"."EM - 201"."QT201-1_OK".CW.ENABLE := True;
   MachineConfig[7]."Unit Process"."EM - 201"."QT201-1_OK".CW.EXIST := True;
   MachineConfig[7]."Unit Process"."EM - 212"."AV212-1".CW.ENABLE := True;
   MachineConfig[7]."Unit Process"."EM - 22X"."AV220-1".CW.ENABLE := True;
   MachineConfig[7]."Unit Process"."EM - 22X"."AV460-1".CW.ENABLE := True;
   MachineConfig[7]."Unit Process"."EM - 22X"."FIT22X-1".CW.ENABLE := True;
   MachineConfig[7]."Unit Process"."EM - 22X"."FIT22X-1".CW.EXIST := false;
   MachineConfig[7]."Unit Process"."EM - 22X"."PIT22X-1".Tag := 'PIT220-1';
   MachineConfig[7]."Unit Process"."EM - 22X"."PIT22X-1".CW.ENABLE := True;
   MachineConfig[7]."Unit Process"."EM - 22X"."QT220-1".CW.ENABLE := True;
   MachineConfig[7]."Unit Process"."EM - 22X"."PCV22X-1".Tag := 'PCV220-1';
   MachineConfig[7]."Unit Process"."EM - 22X"."PCV22X-1".CW.ENABLE := True;
   MachineConfig[7]."Unit Process"."EM - 22X"."PCV22X-1".CW.EXIST := True;
   MachineConfig[7]."Unit Process"."EM - 22X"."QT220-1_OK".CW.ENABLE := True;
   MachineConfig[7]."Unit Process"."EM - 22X"."QT220-1_OK".CW.EXIST := False;
   MachineConfig[7]."Unit Process"."EM - 22X"."LA220-1".CW.ENABLE := True;
   MachineConfig[7]."Unit Process"."EM - 340"."AV340-1".CW.ENABLE := true;
   MachineConfig[7]."Unit Process"."EM - 340"."AV340-2".CW.ENABLE := true;
   MachineConfig[7]."Unit Process"."EM - 340"."AV460-2".CW.ENABLE := true;
   MachineConfig[7]."Unit Process"."EM - 340"."PIS340-1".CW.ENABLE := True;
   MachineConfig[7]."Unit Process"."EM - 340"."PIS340-1".CW.EXIST := True;
   MachineConfig[7]."Unit Dch"."EM - 222"."AV222-1".CW.ENABLE := True;
   MachineConfig[7]."Unit Dch"."EM - 222"."AV222-1".CW.EXIST := True;
   MachineConfig[7]."Unit Dch"."EM - 222"."LS222-1".CW.ENABLE := True;
   MachineConfig[7]."Unit Dch"."EM - 222"."LS222-1".CW.EXIST := True;
   MachineConfig[7]."Unit Dch"."EM - 222"."P222-1".CW.ENABLE := True;
   MachineConfig[7]."Unit Dch"."EM - 222"."P222-1".CW.EXIST := True;
   MachineConfig[7]."Unit Dch"."EM - 222"."TS222-1".CW.ENABLE := true;
   MachineConfig[7]."Unit Dch"."EM - 222"."TT222-1".CW.ENABLE := False;
   MachineConfig[7]."Unit Dch"."EM - 300"."AV301-1".CW.ENABLE := true;
   MachineConfig[7]."Unit Dch"."EM - 300"."AV302-1".CW.ENABLE := true;
   MachineConfig[7]."Unit Dch"."EM - 300"."AV303-1".CW.ENABLE := true;
   MachineConfig[7]."Unit Dch"."EM - 300"."AV304-1".CW.ENABLE := true;
   MachineConfig[7]."Unit Dch"."EM - 300"."AV305-1".CW.ENABLE := true;
   MachineConfig[7]."Unit Dch"."EM - 300"."AV306-1".CW.ENABLE := true;
   MachineConfig[7]."Unit Dch"."EM - 300"."AV320-1".CW.ENABLE := true;
   MachineConfig[7]."Unit Dch"."EM - 300"."AV635-1".CW.ENABLE := true;
   MachineConfig[7]."Unit Dch"."EM - 375"."AV37X-1".CW.ENABLE := True;
   MachineConfig[7]."Unit Dch"."EM - 506"."AV543-1".CW.ENABLE := true;
   MachineConfig[7]."Unit Dch"."EM - 506".IP506a.CW.ENABLE := True;
   MachineConfig[7]."Unit Dch"."EM - 506".AVDCH.CW.ENABLE := True;
   MachineConfig[7].Options."EM - 208"."FIT208-1"."Type" := 2;
   MachineConfig[7].Options."EM - 208"."FIT208-1".Address := 266;
   MachineConfig[7].Options."EM - 208"."FIT208-1".Max := 20000.0;
   MachineConfig[7].Communications."EM - BC-COMM".BCI0 := 8;
   MachineConfig[7].Communications."EM - BC-COMM".BCI1 := 8;
   MachineConfig[7].Communications."EM - BC-COMM".BCI2 := 8;
   MachineConfig[7].Communications."EM - BC-COMM".BCI3 := 8;
   MachineConfig[7].Communications."EM - BC-COMM".BCO0 := 8;
   MachineConfig[7].Communications."EM - BC-COMM".BCO1 := 8;
   MachineConfig[7].Communications."EM - BC-COMM".BCO2 := 8;
   MachineConfig[7].Communications."EM - BC-COMM".BCO3 := 8;
   MachineConfig[7].Communications."EM - BC-COMM".ALARM := 8;
   MachineConfig[8].Machine."Family" := 1;
   MachineConfig[8].Machine.TypeNo := 8;
   MachineConfig[8].Machine.Range := 1;
   MachineConfig[8].Machine.SepType := 1;
   MachineConfig[8].Machine.Frame := 1;
   MachineConfig[8].Machine.DchSystem := 3;
   MachineConfig[8].Machine.Spare_1 := 1;
   MachineConfig[8].Machine.FeedPump := 1;
   MachineConfig[8].Machine.Blending := 1;
   MachineConfig[8].Machine.Recirculation := 1;
   MachineConfig[8].Machine.CoolingRecirculation := 1;
   MachineConfig[8].Machine.Spare_2 := 2;
   MachineConfig[8].Machine.eMotion := 1;
   MachineConfig[8].Machine.ConditionAlert := 1;
   MachineConfig[8].Machine.eWON := 1;
   MachineConfig[8].Machine.ALBufferTank := 1;
   MachineConfig[8]."Unit Sep"."EM - 100"."L-GREEN".CW.ENABLE := True;
   MachineConfig[8]."Unit Sep"."EM - 100"."L-GREEN".CW.EXIST := True;
   MachineConfig[8]."Unit Sep"."EM - 100"."L-YELLOW".CW.ENABLE := True;
   MachineConfig[8]."Unit Sep"."EM - 100"."L-YELLOW".CW.EXIST := True;
   MachineConfig[8]."Unit Sep"."EM - 100".UPS.CW.ENABLE := True;
   MachineConfig[8]."Unit Sep"."EM - 100".UPS.CW.EXIST := True;
   MachineConfig[8]."Unit Sep"."EM - 400"."AV409-1".CW.ENABLE := True;
   MachineConfig[8]."Unit Sep"."EM - 400"."FCV409-1".CW.ENABLE := True;
   MachineConfig[8]."Unit Sep"."EM - 400"."FCV409-1".CW.EXIST := True;
   MachineConfig[8]."Unit Sep"."EM - 400"."FIT409-1".CW.ENABLE := True;
   MachineConfig[8]."Unit Sep"."EM - 400"."FIT409-1".CW.EXIST := True;
   MachineConfig[8]."Unit Sep"."EM - 400"."TT41X-1".CW.ENABLE := True;
   MachineConfig[8]."Unit Sep"."EM - 400"."TT41X-1".CW.EXIST := True;
   MachineConfig[8]."Unit Sep"."EM - 400"."TT41X-1".Address := 142;
   MachineConfig[8]."Unit Sep"."EM - 460"."AV460d-1".CW.ENABLE := True;
   MachineConfig[8]."Unit Sep"."EM - 460"."AV460d-1".FB_OPN_ADD := 214;
   MachineConfig[8]."Unit Sep"."EM - 460"."AV460d-1".FB_CLS_ADD := 215;
   MachineConfig[8]."Unit Sep"."EM - 600"."AV615-1".CW.ENABLE := True;
   MachineConfig[8]."Unit Sep"."EM - 600"."AV615-1".CW.EXIST := True;
   MachineConfig[8]."Unit Sep"."EM - 600"."FIS615-1".CW.ENABLE := True;
   MachineConfig[8]."Unit Sep"."EM - 600"."FIS615-1".CW.EXIST := True;
   MachineConfig[8]."Unit Sep"."EM - 600"."FIS635-1".CW.ENABLE := True;
   MachineConfig[8]."Unit Sep"."EM - 600"."FIS635-1".CW.EXIST := True;
   MachineConfig[8]."Unit Sep"."EM - 701".M701."TYPE" := 1;
   MachineConfig[8]."Unit Sep"."EM - 730".TS730.CW.ENABLE := True;
   MachineConfig[8]."Unit Sep"."EM - 730".TS730.CW.EXIST := True;
   MachineConfig[8]."Unit Sep"."EM - 730".TT731a.CW.ENABLE := True;
   MachineConfig[8]."Unit Sep"."EM - 730".TT731a.CW.EXIST := True;
   MachineConfig[8]."Unit Sep"."EM - 730".TT733.CW.ENABLE := True;
   MachineConfig[8]."Unit Sep"."EM - 730".TT733.CW.EXIST := True;
   MachineConfig[8]."Unit Sep"."EM - 750".YT75X.CW.ENABLE := True;
   MachineConfig[8]."Unit Process"."EM - 201"."AV201-1".CW.ENABLE := True;
   MachineConfig[8]."Unit Process"."EM - 201"."FIT201-1"."Type" := 2;
   MachineConfig[8]."Unit Process"."EM - 201"."FIT201-1".Address := 256;
   MachineConfig[8]."Unit Process"."EM - 201"."FIT201-1".Max := 80000.0;
   MachineConfig[8]."Unit Process"."EM - 201"."LA201-1".CW.ENABLE := true;
   MachineConfig[8]."Unit Process"."EM - 201"."QT201-1".CW.ENABLE := True;
   MachineConfig[8]."Unit Process"."EM - 201"."QT201-1".CW.EXIST := True;
   MachineConfig[8]."Unit Process"."EM - 201"."QT201-1_OK".CW.ENABLE := True;
   MachineConfig[8]."Unit Process"."EM - 201"."QT201-1_OK".CW.EXIST := True;
   MachineConfig[8]."Unit Process"."EM - 212"."AV212-1".CW.ENABLE := True;
   MachineConfig[8]."Unit Process"."EM - 22X"."AV220-1".CW.ENABLE := True;
   MachineConfig[8]."Unit Process"."EM - 22X"."AV460-1".CW.ENABLE := True;
   MachineConfig[8]."Unit Process"."EM - 22X"."PIT22X-1".Tag := 'PIT220-1';
   MachineConfig[8]."Unit Process"."EM - 22X"."PIT22X-1".CW.ENABLE := True;
   MachineConfig[8]."Unit Process"."EM - 22X"."QT220-1".CW.ENABLE := True;
   MachineConfig[8]."Unit Process"."EM - 22X"."PCV22X-1".Tag := 'PCV220-1';
   MachineConfig[8]."Unit Process"."EM - 22X"."PCV22X-1".CW.ENABLE := True;
   MachineConfig[8]."Unit Process"."EM - 22X"."PCV22X-1".CW.EXIST := True;
   MachineConfig[8]."Unit Process"."EM - 22X"."QT220-1_OK".CW.ENABLE := True;
   MachineConfig[8]."Unit Process"."EM - 22X"."QT220-1_OK".CW.EXIST := False;
   MachineConfig[8]."Unit Process"."EM - 22X"."LA220-1".CW.ENABLE := True;
   MachineConfig[8]."Unit Process"."EM - 340"."AV340-1".CW.ENABLE := True;
   MachineConfig[8]."Unit Process"."EM - 340"."AV340-2".CW.ENABLE := True;
   MachineConfig[8]."Unit Process"."EM - 340"."AV460-2".CW.ENABLE := True;
   MachineConfig[8]."Unit Process"."EM - 340"."PIS340-1".CW.ENABLE := True;
   MachineConfig[8]."Unit Process"."EM - 340"."PIS340-1".CW.EXIST := True;
   MachineConfig[8]."Unit Dch"."EM - 222"."AV222-1".CW.ENABLE := True;
   MachineConfig[8]."Unit Dch"."EM - 222"."AV222-1".CW.EXIST := True;
   MachineConfig[8]."Unit Dch"."EM - 222"."LS222-1".CW.ENABLE := True;
   MachineConfig[8]."Unit Dch"."EM - 222"."LS222-1".CW.EXIST := True;
   MachineConfig[8]."Unit Dch"."EM - 222"."P222-1".CW.ENABLE := True;
   MachineConfig[8]."Unit Dch"."EM - 222"."P222-1".CW.EXIST := True;
   MachineConfig[8]."Unit Dch"."EM - 222"."TS222-1".CW.ENABLE := True;
   MachineConfig[8]."Unit Dch"."EM - 222"."TS222-1".CW.EXIST := True;
   MachineConfig[8]."Unit Dch"."EM - 222"."TT222-1".CW.ENABLE := False;
   MachineConfig[8]."Unit Dch"."EM - 300"."AV301-1".CW.ENABLE := true;
   MachineConfig[8]."Unit Dch"."EM - 300"."AV303-1".CW.ENABLE := true;
   MachineConfig[8]."Unit Dch"."EM - 300"."AV304-1".CW.ENABLE := true;
   MachineConfig[8]."Unit Dch"."EM - 300"."AV305-1".CW.ENABLE := true;
   MachineConfig[8]."Unit Dch"."EM - 300"."AV306-1".CW.ENABLE := true;
   MachineConfig[8]."Unit Dch"."EM - 300"."AV320-1".CW.ENABLE := true;
   MachineConfig[8]."Unit Dch"."EM - 300"."AV635-1".CW.ENABLE := true;
   MachineConfig[8]."Unit Dch"."EM - 375"."AV37X-1".CW.ENABLE := true;
   MachineConfig[8]."Unit Dch"."EM - 375"."PT37X-1".CW.ENABLE := True;
   MachineConfig[8]."Unit Dch"."EM - 375"."PT37X-1".CW.EXIST := True;
   MachineConfig[8]."Unit Dch"."EM - 506"."AV543-1".CW.ENABLE := true;
   MachineConfig[8]."Unit Dch"."EM - 506".IP506a.CW.ENABLE := True;
   MachineConfig[8]."Unit Dch"."EM - 506"."PV376-1".CW.ENABLE := true;
   MachineConfig[8]."Unit Dch"."EM - 506"."PV376-2".CW.ENABLE := true;
   MachineConfig[8]."Unit Dch"."EM - 506".AVDCH.CW.ENABLE := true;
   MachineConfig[8].Options."EM - 208"."FIT208-1"."Type" := 2;
   MachineConfig[8].Options."EM - 208"."FIT208-1".Address := 266;
   MachineConfig[8].Options."EM - 208"."FIT208-1".Max := 20000.0;
   MachineConfig[8].Communications."EM - BC-COMM".BCI0 := 8;
   MachineConfig[8].Communications."EM - BC-COMM".BCI1 := 8;
   MachineConfig[8].Communications."EM - BC-COMM".BCI2 := 8;
   MachineConfig[8].Communications."EM - BC-COMM".BCI3 := 8;
   MachineConfig[8].Communications."EM - BC-COMM".BCO0 := 8;
   MachineConfig[8].Communications."EM - BC-COMM".BCO1 := 8;
   MachineConfig[8].Communications."EM - BC-COMM".BCO2 := 8;
   MachineConfig[8].Communications."EM - BC-COMM".BCO3 := 8;
   MachineConfig[8].Communications."EM - BC-COMM".ALARM := 8;
   MachineConfig[9].Machine."Family" := 1;
   MachineConfig[9].Machine.TypeNo := 9;
   MachineConfig[9].Machine.Range := 1;
   MachineConfig[9].Machine.SepType := 1;
   MachineConfig[9].Machine.Frame := 1;
   MachineConfig[9].Machine.DchSystem := 3;
   MachineConfig[9].Machine.Spare_1 := 1;
   MachineConfig[9].Machine.FeedPump := 1;
   MachineConfig[9].Machine.Blending := 1;
   MachineConfig[9].Machine.Recirculation := 1;
   MachineConfig[9].Machine.CoolingRecirculation := 1;
   MachineConfig[9].Machine.Spare_2 := 2;
   MachineConfig[9].Machine.eMotion := 1;
   MachineConfig[9].Machine.ConditionAlert := 1;
   MachineConfig[9].Machine.eWON := 1;
   MachineConfig[9].Machine.ALBufferTank := 1;
   MachineConfig[9]."Unit Sep"."EM - 100"."L-GREEN".CW.ENABLE := True;
   MachineConfig[9]."Unit Sep"."EM - 100"."L-GREEN".CW.EXIST := True;
   MachineConfig[9]."Unit Sep"."EM - 100"."L-YELLOW".CW.ENABLE := True;
   MachineConfig[9]."Unit Sep"."EM - 100"."L-YELLOW".CW.EXIST := True;
   MachineConfig[9]."Unit Sep"."EM - 100".UPS.CW.ENABLE := True;
   MachineConfig[9]."Unit Sep"."EM - 100".UPS.CW.EXIST := True;
   MachineConfig[9]."Unit Sep"."EM - 100"."CA VIB WARN".CW.ENABLE := True;
   MachineConfig[9]."Unit Sep"."EM - 100"."CA VIB ALM".CW.ENABLE := True;
   MachineConfig[9]."Unit Sep"."EM - 100"."CA ERROR".CW.ENABLE := true;
   MachineConfig[9]."Unit Sep"."EM - 100"."CA WD".CW.ENABLE := true;
   MachineConfig[9]."Unit Sep"."EM - 400"."AV409-1".CW.ENABLE := true;
   MachineConfig[9]."Unit Sep"."EM - 400"."FCV409-1".CW.ENABLE := True;
   MachineConfig[9]."Unit Sep"."EM - 400"."FCV409-1".CW.EXIST := True;
   MachineConfig[9]."Unit Sep"."EM - 400"."FIT409-1".CW.ENABLE := True;
   MachineConfig[9]."Unit Sep"."EM - 400"."FIT409-1".CW.EXIST := True;
   MachineConfig[9]."Unit Sep"."EM - 400"."FIT412-1".CW.ENABLE := True;
   MachineConfig[9]."Unit Sep"."EM - 400"."TT41X-1".CW.ENABLE := True;
   MachineConfig[9]."Unit Sep"."EM - 400"."TT41X-1".CW.EXIST := True;
   MachineConfig[9]."Unit Sep"."EM - 400"."TT41X-1".Address := 142;
   MachineConfig[9]."Unit Sep"."EM - 460"."AV460d-1".CW.ENABLE := True;
   MachineConfig[9]."Unit Sep"."EM - 460"."AV460d-1".FB_OPN_ADD := 214;
   MachineConfig[9]."Unit Sep"."EM - 460"."AV460d-1".FB_CLS_ADD := 215;
   MachineConfig[9]."Unit Sep"."EM - 600"."AV615-1".CW.ENABLE := True;
   MachineConfig[9]."Unit Sep"."EM - 600"."FIS615-1".CW.ENABLE := True;
   MachineConfig[9]."Unit Sep"."EM - 600"."FIS615-1".CW.EXIST := True;
   MachineConfig[9]."Unit Sep"."EM - 600"."FIS635-1".CW.ENABLE := True;
   MachineConfig[9]."Unit Sep"."EM - 600"."FIS635-1".CW.EXIST := True;
   MachineConfig[9]."Unit Sep"."EM - 730".TS730.CW.ENABLE := True;
   MachineConfig[9]."Unit Sep"."EM - 730".TS730.CW.EXIST := True;
   MachineConfig[9]."Unit Sep"."EM - 730".TT731a.CW.ENABLE := True;
   MachineConfig[9]."Unit Sep"."EM - 730".TT731a.CW.EXIST := True;
   MachineConfig[9]."Unit Sep"."EM - 730".TT733.CW.ENABLE := True;
   MachineConfig[9]."Unit Sep"."EM - 730".TT733.CW.EXIST := True;
   MachineConfig[9]."Unit Sep"."EM - 750".YT75X.CW.ENABLE := True;
   MachineConfig[9]."Unit Process"."EM - 201"."AV201-1".CW.ENABLE := True;
   MachineConfig[9]."Unit Process"."EM - 201"."FIT201-1"."Type" := 2;
   MachineConfig[9]."Unit Process"."EM - 201"."FIT201-1".Address := 256;
   MachineConfig[9]."Unit Process"."EM - 201"."FIT201-1".Max := 100000.0;
   MachineConfig[9]."Unit Process"."EM - 201"."LA201-1".CW.ENABLE := true;
   MachineConfig[9]."Unit Process"."EM - 201"."QT201-1".CW.ENABLE := True;
   MachineConfig[9]."Unit Process"."EM - 201"."QT201-1".CW.EXIST := True;
   MachineConfig[9]."Unit Process"."EM - 201"."QT201-1_OK".CW.ENABLE := True;
   MachineConfig[9]."Unit Process"."EM - 201"."QT201-1_OK".CW.EXIST := True;
   MachineConfig[9]."Unit Process"."EM - 212"."AV212-1".CW.ENABLE := True;
   MachineConfig[9]."Unit Process"."EM - 22X"."AV220-1".CW.ENABLE := True;
   MachineConfig[9]."Unit Process"."EM - 22X"."AV460-1".CW.ENABLE := True;
   MachineConfig[9]."Unit Process"."EM - 22X"."PIT22X-1".Tag := 'PIT220-1';
   MachineConfig[9]."Unit Process"."EM - 22X"."PIT22X-1".CW.ENABLE := True;
   MachineConfig[9]."Unit Process"."EM - 22X"."PIT22X-1".CW.EXIST := True;
   MachineConfig[9]."Unit Process"."EM - 22X"."QT220-1".CW.ENABLE := True;
   MachineConfig[9]."Unit Process"."EM - 22X"."QT220-1".CW.EXIST := True;
   MachineConfig[9]."Unit Process"."EM - 22X"."PCV22X-1".Tag := 'PCV220-1';
   MachineConfig[9]."Unit Process"."EM - 22X"."PCV22X-1".CW.ENABLE := True;
   MachineConfig[9]."Unit Process"."EM - 22X"."PCV22X-1".CW.EXIST := True;
   MachineConfig[9]."Unit Process"."EM - 22X"."QT220-1_OK".CW.ENABLE := true;
   MachineConfig[9]."Unit Process"."EM - 22X"."QT220-1_OK".CW.EXIST := false;
   MachineConfig[9]."Unit Process"."EM - 22X"."LA220-1".CW.ENABLE := True;
   MachineConfig[9]."Unit Process"."EM - 340"."AV340-1".CW.ENABLE := True;
   MachineConfig[9]."Unit Process"."EM - 340"."AV340-2".CW.ENABLE := True;
   MachineConfig[9]."Unit Process"."EM - 340"."AV460-2".CW.ENABLE := True;
   MachineConfig[9]."Unit Process"."EM - 340"."PIS340-1".CW.ENABLE := True;
   MachineConfig[9]."Unit Process"."EM - 340"."PIS340-1".CW.EXIST := True;
   MachineConfig[9]."Unit Dch"."EM - 222"."AV222-1".CW.ENABLE := True;
   MachineConfig[9]."Unit Dch"."EM - 222"."AV222-1".CW.EXIST := True;
   MachineConfig[9]."Unit Dch"."EM - 222"."LS222-1".CW.ENABLE := True;
   MachineConfig[9]."Unit Dch"."EM - 222"."LS222-1".CW.EXIST := True;
   MachineConfig[9]."Unit Dch"."EM - 222"."P222-1".CW.ENABLE := True;
   MachineConfig[9]."Unit Dch"."EM - 222"."P222-1".CW.EXIST := True;
   MachineConfig[9]."Unit Dch"."EM - 222"."TS222-1".CW.ENABLE := True;
   MachineConfig[9]."Unit Dch"."EM - 222"."TS222-1".CW.EXIST := True;
   MachineConfig[9]."Unit Dch"."EM - 222"."TT222-1".CW.ENABLE := False;
   MachineConfig[9]."Unit Dch"."EM - 222"."TT222-1".CW.EXIST := False;
   MachineConfig[9]."Unit Dch"."EM - 300"."AV301-1".CW.ENABLE := True;
   MachineConfig[9]."Unit Dch"."EM - 300"."AV302-1".CW.ENABLE := True;
   MachineConfig[9]."Unit Dch"."EM - 300"."AV303-1".CW.ENABLE := True;
   MachineConfig[9]."Unit Dch"."EM - 300"."AV304-1".CW.ENABLE := True;
   MachineConfig[9]."Unit Dch"."EM - 300"."AV305-1".CW.ENABLE := True;
   MachineConfig[9]."Unit Dch"."EM - 300"."AV306-1".CW.ENABLE := True;
   MachineConfig[9]."Unit Dch"."EM - 300"."AV320-1".CW.ENABLE := True;
   MachineConfig[9]."Unit Dch"."EM - 375"."AV37X-1".CW.ENABLE := True;
   MachineConfig[9]."Unit Dch"."EM - 375"."PT37X-1".CW.ENABLE := True;
   MachineConfig[9]."Unit Dch"."EM - 375"."PT37X-1".CW.EXIST := True;
   MachineConfig[9]."Unit Dch"."EM - 506"."AV543-1".CW.ENABLE := true;
   MachineConfig[9]."Unit Dch"."EM - 506".IP506a.CW.ENABLE := True;
   MachineConfig[9]."Unit Dch"."EM - 506".IP506a.CW.EXIST := True;
   MachineConfig[9]."Unit Dch"."EM - 506"."PV376-1".CW.ENABLE := True;
   MachineConfig[9]."Unit Dch"."EM - 506"."PV376-2".CW.ENABLE := True;
   MachineConfig[9]."Unit Dch"."EM - 506".AVDCH.CW.ENABLE := True;
   MachineConfig[9].Options."EM - 208"."FIT208-1"."Type" := 2;
   MachineConfig[9].Options."EM - 208"."FIT208-1".Address := 266;
   MachineConfig[9].Options."EM - 208"."FIT208-1".Max := 20000.0;
   MachineConfig[9].Communications."EM - BC-COMM".BCI0 := 8;
   MachineConfig[9].Communications."EM - BC-COMM".BCI1 := 8;
   MachineConfig[9].Communications."EM - BC-COMM".BCI2 := 8;
   MachineConfig[9].Communications."EM - BC-COMM".BCI3 := 8;
   MachineConfig[9].Communications."EM - BC-COMM".BCO0 := 8;
   MachineConfig[9].Communications."EM - BC-COMM".BCO1 := 8;
   MachineConfig[9].Communications."EM - BC-COMM".BCO2 := 8;
   MachineConfig[9].Communications."EM - BC-COMM".BCO3 := 8;
   MachineConfig[9].Communications."EM - BC-COMM".ALARM := 8;
   MachineConfig[10].Machine."Family" := 1;
   MachineConfig[10].Machine.TypeNo := 10;
   MachineConfig[10].Machine.Range := 1;
   MachineConfig[10].Machine.SepType := 1;
   MachineConfig[10].Machine.Frame := 1;
   MachineConfig[10].Machine.DchSystem := 3;
   MachineConfig[10].Machine.Spare_1 := 1;
   MachineConfig[10].Machine.FeedPump := 1;
   MachineConfig[10].Machine.Blending := 1;
   MachineConfig[10].Machine.Recirculation := 1;
   MachineConfig[10].Machine.CoolingRecirculation := 1;
   MachineConfig[10].Machine.Spare_2 := 2;
   MachineConfig[10].Machine.eMotion := 1;
   MachineConfig[10].Machine.ConditionAlert := 1;
   MachineConfig[10].Machine.eWON := 1;
   MachineConfig[10].Machine.ALBufferTank := 1;
   MachineConfig[10]."Unit Sep"."EM - 100"."L-GREEN".CW.ENABLE := True;
   MachineConfig[10]."Unit Sep"."EM - 100"."L-GREEN".CW.EXIST := True;
   MachineConfig[10]."Unit Sep"."EM - 100"."L-YELLOW".CW.ENABLE := True;
   MachineConfig[10]."Unit Sep"."EM - 100"."L-YELLOW".CW.EXIST := True;
   MachineConfig[10]."Unit Sep"."EM - 100".UPS.CW.ENABLE := True;
   MachineConfig[10]."Unit Sep"."EM - 100".UPS.CW.EXIST := True;
   MachineConfig[10]."Unit Sep"."EM - 100"."CA VIB WARN".CW.ENABLE := True;
   MachineConfig[10]."Unit Sep"."EM - 100"."CA VIB ALM".CW.ENABLE := True;
   MachineConfig[10]."Unit Sep"."EM - 100"."CA ERROR".CW.ENABLE := true;
   MachineConfig[10]."Unit Sep"."EM - 100"."CA WD".CW.ENABLE := true;
   MachineConfig[10]."Unit Sep"."EM - 400"."AV409-1".CW.ENABLE := true;
   MachineConfig[10]."Unit Sep"."EM - 400"."FCV409-1".CW.ENABLE := True;
   MachineConfig[10]."Unit Sep"."EM - 400"."FCV409-1".CW.EXIST := True;
   MachineConfig[10]."Unit Sep"."EM - 400"."FIT409-1".CW.ENABLE := True;
   MachineConfig[10]."Unit Sep"."EM - 400"."FIT412-1".CW.ENABLE := True;
   MachineConfig[10]."Unit Sep"."EM - 400"."TT41X-1".CW.ENABLE := True;
   MachineConfig[10]."Unit Sep"."EM - 400"."TT41X-1".CW.EXIST := True;
   MachineConfig[10]."Unit Sep"."EM - 400"."TT41X-1".Address := 142;
   MachineConfig[10]."Unit Sep"."EM - 460"."AV460d-1".CW.ENABLE := True;
   MachineConfig[10]."Unit Sep"."EM - 460"."AV460d-1".FB_OPN_ADD := 214;
   MachineConfig[10]."Unit Sep"."EM - 460"."AV460d-1".FB_CLS_ADD := 215;
   MachineConfig[10]."Unit Sep"."EM - 600"."AV615-1".CW.ENABLE := True;
   MachineConfig[10]."Unit Sep"."EM - 600"."AV615-1".CW.EXIST := True;
   MachineConfig[10]."Unit Sep"."EM - 600"."FIS615-1".CW.ENABLE := True;
   MachineConfig[10]."Unit Sep"."EM - 600"."FIS615-1".CW.EXIST := True;
   MachineConfig[10]."Unit Sep"."EM - 600"."FIS635-1".CW.ENABLE := True;
   MachineConfig[10]."Unit Sep"."EM - 600"."FIS635-1".CW.EXIST := True;
   MachineConfig[10]."Unit Sep"."EM - 730".TS730.CW.ENABLE := True;
   MachineConfig[10]."Unit Sep"."EM - 730".TS730.CW.EXIST := True;
   MachineConfig[10]."Unit Sep"."EM - 730".TT731a.CW.ENABLE := True;
   MachineConfig[10]."Unit Sep"."EM - 730".TT731a.CW.EXIST := True;
   MachineConfig[10]."Unit Sep"."EM - 730".TT733.CW.ENABLE := True;
   MachineConfig[10]."Unit Sep"."EM - 730".TT733.CW.EXIST := True;
   MachineConfig[10]."Unit Sep"."EM - 750".YT75X.CW.ENABLE := True;
   MachineConfig[10]."Unit Process"."EM - 201"."AV201-1".CW.ENABLE := True;
   MachineConfig[10]."Unit Process"."EM - 201"."FIT201-1"."Type" := 2;
   MachineConfig[10]."Unit Process"."EM - 201"."FIT201-1".Address := 256;
   MachineConfig[10]."Unit Process"."EM - 201"."FIT201-1".Max := 100000.0;
   MachineConfig[10]."Unit Process"."EM - 201"."LA201-1".CW.ENABLE := true;
   MachineConfig[10]."Unit Process"."EM - 201"."QT201-1".CW.ENABLE := True;
   MachineConfig[10]."Unit Process"."EM - 201"."QT201-1".CW.EXIST := True;
   MachineConfig[10]."Unit Process"."EM - 201"."QT201-1_OK".CW.ENABLE := True;
   MachineConfig[10]."Unit Process"."EM - 201"."QT201-1_OK".CW.EXIST := True;
   MachineConfig[10]."Unit Process"."EM - 212"."AV212-1".CW.ENABLE := True;
   MachineConfig[10]."Unit Process"."EM - 22X"."AV220-1".CW.ENABLE := True;
   MachineConfig[10]."Unit Process"."EM - 22X"."AV460-1".CW.ENABLE := True;
   MachineConfig[10]."Unit Process"."EM - 22X"."PIT22X-1".Tag := 'PIT220-1';
   MachineConfig[10]."Unit Process"."EM - 22X"."PIT22X-1".CW.ENABLE := True;
   MachineConfig[10]."Unit Process"."EM - 22X"."PIT22X-1".CW.EXIST := True;
   MachineConfig[10]."Unit Process"."EM - 22X"."QT220-1".Tag := 'QT220-1';
   MachineConfig[10]."Unit Process"."EM - 22X"."QT220-1".CW.ENABLE := True;
   MachineConfig[10]."Unit Process"."EM - 22X"."PCV22X-1".Tag := 'PCV220-1';
   MachineConfig[10]."Unit Process"."EM - 22X"."PCV22X-1".CW.ENABLE := True;
   MachineConfig[10]."Unit Process"."EM - 22X"."QT220-1_OK".CW.INPUT := True;
   MachineConfig[10]."Unit Process"."EM - 22X"."QT220-1_OK".CW.EXIST := False;
   MachineConfig[10]."Unit Process"."EM - 22X"."LA220-1".CW.ENABLE := True;
   MachineConfig[10]."Unit Process"."EM - 340"."AV340-1".CW.ENABLE := True;
   MachineConfig[10]."Unit Process"."EM - 340"."AV340-2".CW.ENABLE := True;
   MachineConfig[10]."Unit Process"."EM - 340"."AV460-2".CW.ENABLE := True;
   MachineConfig[10]."Unit Process"."EM - 340"."PIS340-1".CW.ENABLE := True;
   MachineConfig[10]."Unit Process"."EM - 340"."PIS340-1".CW.EXIST := True;
   MachineConfig[10]."Unit Dch"."EM - 222"."AV222-1".CW.ENABLE := True;
   MachineConfig[10]."Unit Dch"."EM - 222"."AV222-1".CW.EXIST := True;
   MachineConfig[10]."Unit Dch"."EM - 222"."LS222-1".CW.ENABLE := True;
   MachineConfig[10]."Unit Dch"."EM - 222"."LS222-1".CW.EXIST := True;
   MachineConfig[10]."Unit Dch"."EM - 222"."P222-1".CW.ENABLE := True;
   MachineConfig[10]."Unit Dch"."EM - 222"."P222-1".CW.EXIST := True;
   MachineConfig[10]."Unit Dch"."EM - 222"."TS222-1".CW.ENABLE := True;
   MachineConfig[10]."Unit Dch"."EM - 222"."TS222-1".CW.EXIST := True;
   MachineConfig[10]."Unit Dch"."EM - 300"."AV301-1".CW.ENABLE := True;
   MachineConfig[10]."Unit Dch"."EM - 300"."AV302-1".CW.ENABLE := True;
   MachineConfig[10]."Unit Dch"."EM - 300"."AV303-1".CW.ENABLE := True;
   MachineConfig[10]."Unit Dch"."EM - 300"."AV304-1".CW.ENABLE := True;
   MachineConfig[10]."Unit Dch"."EM - 300"."AV305-1".CW.ENABLE := True;
   MachineConfig[10]."Unit Dch"."EM - 300"."AV306-1".CW.ENABLE := True;
   MachineConfig[10]."Unit Dch"."EM - 300"."AV320-1".CW.ENABLE := True;
   MachineConfig[10]."Unit Dch"."EM - 300"."AV635-1".CW.ENABLE := True;
   MachineConfig[10]."Unit Dch"."EM - 375"."AV37X-1".CW.ENABLE := True;
   MachineConfig[10]."Unit Dch"."EM - 375"."PT37X-1".CW.ENABLE := True;
   MachineConfig[10]."Unit Dch"."EM - 375"."PT37X-1".CW.EXIST := True;
   MachineConfig[10]."Unit Dch"."EM - 506"."AV543-1".CW.ENABLE := true;
   MachineConfig[10]."Unit Dch"."EM - 506".IP506a.CW.ENABLE := True;
   MachineConfig[10]."Unit Dch"."EM - 506".IP506a.CW.EXIST := True;
   MachineConfig[10]."Unit Dch"."EM - 506"."PV376-1".CW.ENABLE := True;
   MachineConfig[10]."Unit Dch"."EM - 506"."PV376-2".CW.ENABLE := True;
   MachineConfig[10]."Unit Dch"."EM - 506".AVDCH.CW.ENABLE := True;
   MachineConfig[10].Options."EM - 208"."FIT208-1"."Type" := 2;
   MachineConfig[10].Options."EM - 208"."FIT208-1".Address := 266;
   MachineConfig[10].Options."EM - 208"."FIT208-1".Max := 20000.0;
   MachineConfig[10].Communications."EM - BC-COMM".BCI0 := 8;
   MachineConfig[10].Communications."EM - BC-COMM".BCI1 := 8;
   MachineConfig[10].Communications."EM - BC-COMM".BCI2 := 8;
   MachineConfig[10].Communications."EM - BC-COMM".BCI3 := 8;
   MachineConfig[10].Communications."EM - BC-COMM".BCO0 := 8;
   MachineConfig[10].Communications."EM - BC-COMM".BCO1 := 8;
   MachineConfig[10].Communications."EM - BC-COMM".BCO2 := 8;
   MachineConfig[10].Communications."EM - BC-COMM".BCO3 := 8;
   MachineConfig[10].Communications."EM - BC-COMM".ALARM := 8;
   MachineConfig[11].Machine."Family" := 1;
   MachineConfig[11].Machine.TypeNo := 11;
   MachineConfig[11].Machine.Range := 1;
   MachineConfig[11].Machine.SepType := 1;
   MachineConfig[11].Machine.Frame := 2;
   MachineConfig[11].Machine.DchSystem := 3;
   MachineConfig[11].Machine.Spare_1 := 1;
   MachineConfig[11].Machine.FeedPump := 1;
   MachineConfig[11].Machine.Blending := 1;
   MachineConfig[11].Machine.Recirculation := 1;
   MachineConfig[11].Machine.CoolingRecirculation := 1;
   MachineConfig[11].Machine.Spare_2 := 2;
   MachineConfig[11].Machine.eMotion := 1;
   MachineConfig[11].Machine.ConditionAlert := 1;
   MachineConfig[11].Machine.eWON := 1;
   MachineConfig[11].Machine.ALBufferTank := 1;
   MachineConfig[11]."Unit Sep"."EM - 100"."L-GREEN".CW.ENABLE := True;
   MachineConfig[11]."Unit Sep"."EM - 100"."L-GREEN".CW.EXIST := True;
   MachineConfig[11]."Unit Sep"."EM - 100"."L-YELLOW".CW.ENABLE := True;
   MachineConfig[11]."Unit Sep"."EM - 100"."L-YELLOW".CW.EXIST := True;
   MachineConfig[11]."Unit Sep"."EM - 100".UPS.CW.ENABLE := True;
   MachineConfig[11]."Unit Sep"."EM - 100".UPS.CW.EXIST := True;
   MachineConfig[11]."Unit Sep"."EM - 100"."CA VIB WARN".CW.ENABLE := True;
   MachineConfig[11]."Unit Sep"."EM - 100"."CA VIB ALM".CW.ENABLE := true;
   MachineConfig[11]."Unit Sep"."EM - 100"."CA ERROR".CW.ENABLE := true;
   MachineConfig[11]."Unit Sep"."EM - 100"."CA WD".CW.ENABLE := true;
   MachineConfig[11]."Unit Sep"."EM - 400"."AV409-1".CW.FORCE := TRUE;
   MachineConfig[11]."Unit Sep"."EM - 400"."FCV409-1".CW.ENABLE := True;
   MachineConfig[11]."Unit Sep"."EM - 400"."FCV409-1".CW.EXIST := True;
   MachineConfig[11]."Unit Sep"."EM - 400"."FIS412-1".CW.ENABLE := True;
   MachineConfig[11]."Unit Sep"."EM - 400"."FIT409-1".CW.ENABLE := True;
   MachineConfig[11]."Unit Sep"."EM - 400"."FIT409-1".CW.EXIST := True;
   MachineConfig[11]."Unit Sep"."EM - 400"."FIT412-1".CW.ENABLE := True;
   MachineConfig[11]."Unit Sep"."EM - 400"."TT411-1".CW.ENABLE := True;
   MachineConfig[11]."Unit Sep"."EM - 400"."TT41X-1".Tag := 'TT412-1';
   MachineConfig[11]."Unit Sep"."EM - 400"."TT41X-1".CW.ENABLE := True;
   MachineConfig[11]."Unit Sep"."EM - 400"."TT41X-1".CW.EXIST := True;
   MachineConfig[11]."Unit Sep"."EM - 400"."TT41X-1".Address := 142;
   MachineConfig[11]."Unit Sep"."EM - 420".FS421a.CW.ENABLE := true;
   MachineConfig[11]."Unit Sep"."EM - 420".FS421b.CW.ENABLE := true;
   MachineConfig[11]."Unit Sep"."EM - 420".LS422a.CW.ENABLE := true;
   MachineConfig[11]."Unit Sep"."EM - 420"."LS42X(b)".CW.ENABLE := true;
   MachineConfig[11]."Unit Sep"."EM - 420"."LS422-1".CW.ENABLE := true;
   MachineConfig[11]."Unit Sep"."EM - 420"."P403-1".CW.ENABLE := True;
   MachineConfig[11]."Unit Sep"."EM - 420"."P421-1".CW.ENABLE := True;
   MachineConfig[11]."Unit Sep"."EM - 420"."PV421-1".CW.ENABLE := True;
   MachineConfig[11]."Unit Sep"."EM - 460"."AV460d-1".CW.ENABLE := True;
   MachineConfig[11]."Unit Sep"."EM - 460"."AV460d-1".FB_OPN_ADD := 214;
   MachineConfig[11]."Unit Sep"."EM - 460"."AV460d-1".FB_CLS_ADD := 215;
   MachineConfig[11]."Unit Sep"."EM - 600"."AV615-1".CW.ENABLE := True;
   MachineConfig[11]."Unit Sep"."EM - 600"."FIS615-1".CW.ENABLE := True;
   MachineConfig[11]."Unit Sep"."EM - 600"."FIS615-1".CW.EXIST := True;
   MachineConfig[11]."Unit Sep"."EM - 600"."FIS635-1".CW.ENABLE := True;
   MachineConfig[11]."Unit Sep"."EM - 600"."FIS635-1".CW.EXIST := True;
   MachineConfig[11]."Unit Sep"."EM - 730".TS730.CW.ENABLE := True;
   MachineConfig[11]."Unit Sep"."EM - 730".TS730.CW.EXIST := True;
   MachineConfig[11]."Unit Sep"."EM - 730".TT730a.CW.ENABLE := True;
   MachineConfig[11]."Unit Sep"."EM - 730".TT730a.CW.EXIST := True;
   MachineConfig[11]."Unit Sep"."EM - 730".TT730b.CW.ENABLE := True;
   MachineConfig[11]."Unit Sep"."EM - 730".TT731a.CW.ENABLE := True;
   MachineConfig[11]."Unit Sep"."EM - 730".TT734.CW.ENABLE := True;
   MachineConfig[11]."Unit Sep"."EM - 750".YT75X.CW.ENABLE := True;
   MachineConfig[11]."Unit Process"."EM - 201"."AV201-1".CW.ENABLE := True;
   MachineConfig[11]."Unit Process"."EM - 201"."FIT201-1"."Type" := 2;
   MachineConfig[11]."Unit Process"."EM - 201"."FIT201-1".Address := 256;
   MachineConfig[11]."Unit Process"."EM - 201"."FIT201-1".Max := 100000.0;
   MachineConfig[11]."Unit Process"."EM - 201"."LA201-1".CW.ENABLE := true;
   MachineConfig[11]."Unit Process"."EM - 201"."QT201-1".CW.ENABLE := True;
   MachineConfig[11]."Unit Process"."EM - 201"."QT201-1".CW.EXIST := True;
   MachineConfig[11]."Unit Process"."EM - 201"."QT201-1_OK".CW.ENABLE := True;
   MachineConfig[11]."Unit Process"."EM - 201"."QT201-1_OK".CW.EXIST := True;
   MachineConfig[11]."Unit Process"."EM - 212"."AV212-1".CW.ENABLE := True;
   MachineConfig[11]."Unit Process"."EM - 22X"."AV220-1".CW.ENABLE := True;
   MachineConfig[11]."Unit Process"."EM - 22X"."AV460-1".CW.ENABLE := True;
   MachineConfig[11]."Unit Process"."EM - 22X"."PIT22X-1".Tag := 'PIT220-1';
   MachineConfig[11]."Unit Process"."EM - 22X"."PIT22X-1".CW.ENABLE := True;
   MachineConfig[11]."Unit Process"."EM - 22X"."QT220-1".Tag := 'QT220-1';
   MachineConfig[11]."Unit Process"."EM - 22X"."QT220-1".CW.ENABLE := True;
   MachineConfig[11]."Unit Process"."EM - 22X"."PCV22X-1".Tag := 'PCV220-1';
   MachineConfig[11]."Unit Process"."EM - 22X"."PCV22X-1".CW.ENABLE := True;
   MachineConfig[11]."Unit Process"."EM - 22X"."QT220-1_OK".CW.ENABLE := True;
   MachineConfig[11]."Unit Process"."EM - 22X"."QT220-1_OK".CW.EXIST := False;
   MachineConfig[11]."Unit Process"."EM - 22X"."LA220-1".CW.ENABLE := True;
   MachineConfig[11]."Unit Process"."EM - 340"."AV340-1".CW.ENABLE := True;
   MachineConfig[11]."Unit Process"."EM - 340"."AV340-2".CW.ENABLE := True;
   MachineConfig[11]."Unit Process"."EM - 340"."AV460-2".CW.ENABLE := True;
   MachineConfig[11]."Unit Process"."EM - 340"."PIS340-1".CW.ENABLE := True;
   MachineConfig[11]."Unit Process"."EM - 340"."PIS340-1".CW.EXIST := True;
   MachineConfig[11]."Unit Dch"."EM - 222"."AV222-1".CW.ENABLE := True;
   MachineConfig[11]."Unit Dch"."EM - 222"."AV222-1".CW.EXIST := True;
   MachineConfig[11]."Unit Dch"."EM - 222"."LS222-1".CW.ENABLE := True;
   MachineConfig[11]."Unit Dch"."EM - 222"."LS222-1".CW.EXIST := True;
   MachineConfig[11]."Unit Dch"."EM - 222"."P222-1".CW.ENABLE := True;
   MachineConfig[11]."Unit Dch"."EM - 222"."P222-1".CW.EXIST := True;
   MachineConfig[11]."Unit Dch"."EM - 222"."TS222-1".CW.ENABLE := True;
   MachineConfig[11]."Unit Dch"."EM - 222"."TS222-1".CW.EXIST := True;
   MachineConfig[11]."Unit Dch"."EM - 300"."AV301-1".CW.ENABLE := True;
   MachineConfig[11]."Unit Dch"."EM - 300"."AV302-1".CW.ENABLE := True;
   MachineConfig[11]."Unit Dch"."EM - 300"."AV303-1".CW.ENABLE := True;
   MachineConfig[11]."Unit Dch"."EM - 300"."AV304-1".CW.ENABLE := True;
   MachineConfig[11]."Unit Dch"."EM - 300"."AV305-1".CW.ENABLE := True;
   MachineConfig[11]."Unit Dch"."EM - 300"."AV306-1".CW.ENABLE := True;
   MachineConfig[11]."Unit Dch"."EM - 300"."AV320-1".CW.ENABLE := True;
   MachineConfig[11]."Unit Dch"."EM - 300"."AV635-1".CW.ENABLE := True;
   MachineConfig[11]."Unit Dch"."EM - 375"."AV37X-1".CW.ENABLE := True;
   MachineConfig[11]."Unit Dch"."EM - 375"."PT37X-1".CW.ENABLE := True;
   MachineConfig[11]."Unit Dch"."EM - 375"."PT37X-1".CW.EXIST := True;
   MachineConfig[11]."Unit Dch"."EM - 506"."AV543-1".CW.ENABLE := true;
   MachineConfig[11]."Unit Dch"."EM - 506".IP506a.CW.ENABLE := True;
   MachineConfig[11]."Unit Dch"."EM - 506".IP506a.CW.EXIST := True;
   MachineConfig[11]."Unit Dch"."EM - 506"."PV376-1".CW.ENABLE := True;
   MachineConfig[11]."Unit Dch"."EM - 506"."PV376-2".CW.ENABLE := True;
   MachineConfig[11]."Unit Dch"."EM - 506".AVDCH.CW.ENABLE := True;
   MachineConfig[11].Options."EM - 208"."FIT208-1"."Type" := 2;
   MachineConfig[11].Options."EM - 208"."FIT208-1".Address := 266;
   MachineConfig[11].Options."EM - 208"."FIT208-1".Max := 20000.0;
   MachineConfig[11].Communications."EM - BC-COMM".BCI0 := 8;
   MachineConfig[11].Communications."EM - BC-COMM".BCI1 := 8;
   MachineConfig[11].Communications."EM - BC-COMM".BCI2 := 8;
   MachineConfig[11].Communications."EM - BC-COMM".BCI3 := 8;
   MachineConfig[11].Communications."EM - BC-COMM".BCO0 := 8;
   MachineConfig[11].Communications."EM - BC-COMM".BCO1 := 8;
   MachineConfig[11].Communications."EM - BC-COMM".BCO2 := 8;
   MachineConfig[11].Communications."EM - BC-COMM".BCO3 := 8;
   MachineConfig[11].Communications."EM - BC-COMM".ALARM := 8;
   MachineConfig[12].Machine."Family" := 1;
   MachineConfig[12].Machine.TypeNo := 12;
   MachineConfig[12].Machine.Range := 1;
   MachineConfig[12].Machine.SepType := 1;
   MachineConfig[12].Machine.Frame := 2;
   MachineConfig[12].Machine.DchSystem := 3;
   MachineConfig[12].Machine.Spare_1 := 1;
   MachineConfig[12].Machine.FeedPump := 1;
   MachineConfig[12].Machine.Blending := 1;
   MachineConfig[12].Machine.Recirculation := 1;
   MachineConfig[12].Machine.CoolingRecirculation := 1;
   MachineConfig[12].Machine.Spare_2 := 2;
   MachineConfig[12].Machine.eMotion := 1;
   MachineConfig[12].Machine.ConditionAlert := 1;
   MachineConfig[12].Machine.eWON := 1;
   MachineConfig[12].Machine.ALBufferTank := 1;
   MachineConfig[12]."Unit Sep"."EM - 100"."L-GREEN".CW.ENABLE := TRUE;
   MachineConfig[12]."Unit Sep"."EM - 100"."L-YELLOW".CW.ENABLE := TRUE;
   MachineConfig[12]."Unit Sep"."EM - 100"."L-RED".CW.ENABLE := TRUE;
   MachineConfig[12]."Unit Sep"."EM - 100"."L-BUZZ".CW.ENABLE := TRUE;
   MachineConfig[12]."Unit Sep"."EM - 100".EMS.CW.ENABLE := TRUE;
   MachineConfig[12]."Unit Sep"."EM - 100".UPS.CW.ENABLE := True;
   MachineConfig[12]."Unit Sep"."EM - 100".UPS.CW.EXIST := True;
   MachineConfig[12]."Unit Sep"."EM - 100"."CA VIB WARN".CW.ENABLE := True;
   MachineConfig[12]."Unit Sep"."EM - 100"."CA VIB ALM".CW.ENABLE := true;
   MachineConfig[12]."Unit Sep"."EM - 100"."CA ERROR".CW.ENABLE := true;
   MachineConfig[12]."Unit Sep"."EM - 100"."CA WD".CW.ENABLE := true;
   MachineConfig[12]."Unit Sep"."EM - 400"."AV409-1".CW.ENABLE := TRUE;
   MachineConfig[12]."Unit Sep"."EM - 400"."FCV409-1".CW.ENABLE := True;
   MachineConfig[12]."Unit Sep"."EM - 400"."FCV409-1".CW.EXIST := True;
   MachineConfig[12]."Unit Sep"."EM - 400"."FIS409-1".CW.ENABLE := TRUE;
   MachineConfig[12]."Unit Sep"."EM - 400"."FIS412-1".CW.ENABLE := True;
   MachineConfig[12]."Unit Sep"."EM - 400"."FIS412-1".CW.EXIST := True;
   MachineConfig[12]."Unit Sep"."EM - 400"."FIT409-1".CW.ENABLE := True;
   MachineConfig[12]."Unit Sep"."EM - 400"."FIT409-1".CW.EXIST := True;
   MachineConfig[12]."Unit Sep"."EM - 400"."FIT412-1".CW.ENABLE := True;
   MachineConfig[12]."Unit Sep"."EM - 400"."FIT412-1".CW.EXIST := True;
   MachineConfig[12]."Unit Sep"."EM - 400"."TT411-1".CW.ENABLE := True;
   MachineConfig[12]."Unit Sep"."EM - 400"."TT411-1".CW.EXIST := True;
   MachineConfig[12]."Unit Sep"."EM - 400"."TT41X-1".Tag := 'TT412-1';
   MachineConfig[12]."Unit Sep"."EM - 400"."TT41X-1".CW.ENABLE := True;
   MachineConfig[12]."Unit Sep"."EM - 400"."TT41X-1".CW.EXIST := True;
   MachineConfig[12]."Unit Sep"."EM - 400"."TT41X-1".Address := 142;
   MachineConfig[12]."Unit Sep"."EM - 420".FS421a.CW.ENABLE := True;
   MachineConfig[12]."Unit Sep"."EM - 420".FS421a.CW.EXIST := True;
   MachineConfig[12]."Unit Sep"."EM - 420".FS421b.CW.ENABLE := True;
   MachineConfig[12]."Unit Sep"."EM - 420".FS421b.CW.EXIST := True;
   MachineConfig[12]."Unit Sep"."EM - 420".LS422a.CW.ENABLE := TRUE;
   MachineConfig[12]."Unit Sep"."EM - 420"."LS42X(b)".CW.ENABLE := TRUE;
   MachineConfig[12]."Unit Sep"."EM - 420"."LS422-1".CW.ENABLE := TRUE;
   MachineConfig[12]."Unit Sep"."EM - 420"."P403-1".TAG := 'P403-1';
   MachineConfig[12]."Unit Sep"."EM - 420"."P403-1".CW.ENABLE := TRUE;
   MachineConfig[12]."Unit Sep"."EM - 420"."P421-1".CW.ENABLE := TRUE;
   MachineConfig[12]."Unit Sep"."EM - 420"."PV421-1".CW.ENABLE := TRUE;
   MachineConfig[12]."Unit Sep"."EM - 460"."AV460d-1".CW.ENABLE := TRUE;
   MachineConfig[12]."Unit Sep"."EM - 460"."AV460d-1".FB_OPN_ADD := 214;
   MachineConfig[12]."Unit Sep"."EM - 460"."AV460d-1".FB_CLS_ADD := 215;
   MachineConfig[12]."Unit Sep"."EM - 600"."AV615-1".CW.ENABLE := True;
   MachineConfig[12]."Unit Sep"."EM - 600"."FIS615-1".CW.ENABLE := TRUE;
   MachineConfig[12]."Unit Sep"."EM - 600"."FIS635-1".CW.ENABLE := TRUE;
   MachineConfig[12]."Unit Sep"."EM - 730".TS730.CW.ENABLE := True;
   MachineConfig[12]."Unit Sep"."EM - 730".TS730.CW.EXIST := True;
   MachineConfig[12]."Unit Sep"."EM - 730".TT730a.CW.ENABLE := True;
   MachineConfig[12]."Unit Sep"."EM - 730".TT730a.CW.EXIST := True;
   MachineConfig[12]."Unit Sep"."EM - 730".TT730b.CW.ENABLE := True;
   MachineConfig[12]."Unit Sep"."EM - 730".TT730b.CW.EXIST := True;
   MachineConfig[12]."Unit Sep"."EM - 730".TT731a.CW.ENABLE := True;
   MachineConfig[12]."Unit Sep"."EM - 730".TT731a.CW.EXIST := True;
   MachineConfig[12]."Unit Sep"."EM - 730".TT734.CW.ENABLE := True;
   MachineConfig[12]."Unit Sep"."EM - 730".TT734.CW.EXIST := True;
   MachineConfig[12]."Unit Sep"."EM - 740"."P+F PS".CW.ENABLE := TRUE;
   MachineConfig[12]."Unit Sep"."EM - 740"."P+F OS".CW.ENABLE := TRUE;
   MachineConfig[12]."Unit Sep"."EM - 740"."P+F ERROR".CW.ENABLE := TRUE;
   MachineConfig[12]."Unit Sep"."EM - 750".YT75X.CW.ENABLE := True;
   MachineConfig[12]."Unit Process"."EM - 201"."AV201-1".CW.ENABLE := TRUE;
   MachineConfig[12]."Unit Process"."EM - 201"."FIT201-1"."Type" := 2;
   MachineConfig[12]."Unit Process"."EM - 201"."FIT201-1".Address := 256;
   MachineConfig[12]."Unit Process"."EM - 201"."FIT201-1".Max := 100000.0;
   MachineConfig[12]."Unit Process"."EM - 201"."LA201-1".CW.ENABLE := true;
   MachineConfig[12]."Unit Process"."EM - 201"."QT201-1".CW.ENABLE := TRUE;
   MachineConfig[12]."Unit Process"."EM - 201"."QT201-1".CW.EXIST := TRUE;
   MachineConfig[12]."Unit Process"."EM - 201"."TT201-1".CW.EXIST := FALSE;
   MachineConfig[12]."Unit Process"."EM - 201"."QT201-1_OK".CW.ENABLE := True;
   MachineConfig[12]."Unit Process"."EM - 201"."QT201-1_OK".CW.EXIST := True;
   MachineConfig[12]."Unit Process"."EM - 212"."AV212-1".CW.ENABLE := True;
   MachineConfig[12]."Unit Process"."EM - 22X"."AV220-1".CW.ENABLE := True;
   MachineConfig[12]."Unit Process"."EM - 22X"."AV460-1".CW.ENABLE := True;
   MachineConfig[12]."Unit Process"."EM - 22X"."QT220-1".CW.ENABLE := True;
   MachineConfig[12]."Unit Process"."EM - 22X"."QT220-1_OK".CW.ENABLE := True;
   MachineConfig[12]."Unit Process"."EM - 22X"."QT220-1_OK".CW.EXIST := False;
   MachineConfig[12]."Unit Process"."EM - 22X"."LA220-1".CW.ENABLE := True;
   MachineConfig[12]."Unit Process"."EM - 340"."AV340-1".CW.ENABLE := TRUE;
   MachineConfig[12]."Unit Process"."EM - 340"."AV340-2".CW.ENABLE := TRUE;
   MachineConfig[12]."Unit Process"."EM - 340"."AV460-2".CW.ENABLE := TRUE;
   MachineConfig[12]."Unit Process"."EM - 340"."PIS340-1".CW.ENABLE := TRUE;
   MachineConfig[12]."Unit Dch"."EM - 222"."AV222-1".CW.ENABLE := true;
   MachineConfig[12]."Unit Dch"."EM - 222"."LS222-1".CW.ENABLE := TRUE;
   MachineConfig[12]."Unit Dch"."EM - 222"."P222-1".CW.ENABLE := True;
   MachineConfig[12]."Unit Dch"."EM - 222"."P222-1".CW.EXIST := True;
   MachineConfig[12]."Unit Dch"."EM - 222"."TS222-1".CW.ENABLE := true;
   MachineConfig[12]."Unit Dch"."EM - 222"."TT222-1".CW.ENABLE := TRUE;
   MachineConfig[12]."Unit Dch"."EM - 222"."TT222-1".CW.EXIST := FALSE;
   MachineConfig[12]."Unit Dch"."EM - 300"."AV301-1".CW.ENABLE := TRUE;
   MachineConfig[12]."Unit Dch"."EM - 300"."AV302-1".CW.ENABLE := TRUE;
   MachineConfig[12]."Unit Dch"."EM - 300"."AV303-1".CW.ENABLE := TRUE;
   MachineConfig[12]."Unit Dch"."EM - 300"."AV304-1".CW.ENABLE := TRUE;
   MachineConfig[12]."Unit Dch"."EM - 300"."AV305-1".CW.ENABLE := TRUE;
   MachineConfig[12]."Unit Dch"."EM - 300"."AV306-1".CW.ENABLE := TRUE;
   MachineConfig[12]."Unit Dch"."EM - 300"."AV320-1".CW.ENABLE := TRUE;
   MachineConfig[12]."Unit Dch"."EM - 300"."AV635-1".CW.ENABLE := TRUE;
   MachineConfig[12]."Unit Dch"."EM - 375"."AV37X-1".CW.ENABLE := TRUE;
   MachineConfig[12]."Unit Dch"."EM - 375"."PT37X-1".CW.ENABLE := TRUE;
   MachineConfig[12]."Unit Dch"."EM - 506"."AV543-1".CW.ENABLE := TRUE;
   MachineConfig[12]."Unit Dch"."EM - 506".IP506a.CW.ENABLE := TRUE;
   MachineConfig[12]."Unit Dch"."EM - 506"."PV376-1".CW.ENABLE := TRUE;
   MachineConfig[12]."Unit Dch"."EM - 506"."PV376-2".CW.ENABLE := TRUE;
   MachineConfig[12]."Unit Dch"."EM - 506".AVDCH.CW.ENABLE := TRUE;
   MachineConfig[12].Options."EM - 208"."FIT208-1"."Type" := 2;
   MachineConfig[12].Options."EM - 208"."FIT208-1".Address := 266;
   MachineConfig[12].Options."EM - 208"."FIT208-1".Max := 20000.0;
   MachineConfig[12].Communications."EM - BC-COMM".BCI0 := 8;
   MachineConfig[12].Communications."EM - BC-COMM".BCI1 := 8;
   MachineConfig[12].Communications."EM - BC-COMM".BCI2 := 8;
   MachineConfig[12].Communications."EM - BC-COMM".BCI3 := 8;
   MachineConfig[12].Communications."EM - BC-COMM".BCO0 := 8;
   MachineConfig[12].Communications."EM - BC-COMM".BCO1 := 8;
   MachineConfig[12].Communications."EM - BC-COMM".BCO2 := 8;
   MachineConfig[12].Communications."EM - BC-COMM".BCO3 := 8;
   MachineConfig[12].Communications."EM - BC-COMM".ALARM := 8;
   MachineConfig[13].Machine."Family" := 1;
   MachineConfig[13].Machine.TypeNo := 13;
   MachineConfig[13].Machine.Range := 1;
   MachineConfig[13].Machine.SepType := 1;
   MachineConfig[13].Machine.Frame := 2;
   MachineConfig[13].Machine.DchSystem := 3;
   MachineConfig[13].Machine.Spare_1 := 1;
   MachineConfig[13].Machine.FeedPump := 1;
   MachineConfig[13].Machine.Blending := 1;
   MachineConfig[13].Machine.Recirculation := 1;
   MachineConfig[13].Machine.CoolingRecirculation := 1;
   MachineConfig[13].Machine.Spare_2 := 2;
   MachineConfig[13].Machine.eMotion := 1;
   MachineConfig[13].Machine.ConditionAlert := 1;
   MachineConfig[13].Machine.eWON := 1;
   MachineConfig[13]."Unit Sep"."EM - 100".UPS.CW.EXIST := True;
   MachineConfig[13]."Unit Sep"."EM - 100"."CA VIB WARN".CW.ENABLE := True;
   MachineConfig[13]."Unit Sep"."EM - 100"."CA VIB ALM".CW.ENABLE := True;
   MachineConfig[13]."Unit Sep"."EM - 100"."CA ERROR".CW.ENABLE := True;
   MachineConfig[13]."Unit Sep"."EM - 100"."CA WD".CW.ENABLE := True;
   MachineConfig[13]."Unit Sep"."EM - 400"."AV409-1".CW.ENABLE := TRUE;
   MachineConfig[13]."Unit Sep"."EM - 400"."FCV409-1".CW.ENABLE := True;
   MachineConfig[13]."Unit Sep"."EM - 400"."FIT409-1".CW.ENABLE := True;
   MachineConfig[13]."Unit Sep"."EM - 400"."TT411-1".CW.ENABLE := True;
   MachineConfig[13]."Unit Sep"."EM - 400"."TT41X-1".Tag := 'TT412-1';
   MachineConfig[13]."Unit Sep"."EM - 400"."TT41X-1".CW.ENABLE := True;
   MachineConfig[13]."Unit Sep"."EM - 400"."TT41X-1".CW.EXIST := True;
   MachineConfig[13]."Unit Sep"."EM - 420"."LS42X(b)".Tag := 'LS423';
   MachineConfig[13]."Unit Sep"."EM - 420"."LS42X(b)".CW.ENABLE := True;
   MachineConfig[13]."Unit Sep"."EM - 420"."LS42X(b)".CW.EXIST := True;
   MachineConfig[13]."Unit Sep"."EM - 420"."P421-1".CW.ENABLE := True;
   MachineConfig[13]."Unit Sep"."EM - 420"."PS421-1".CW.ENABLE := True;
   MachineConfig[13]."Unit Sep"."EM - 420"."SV421-1".CW.ENABLE := True;
   MachineConfig[13]."Unit Sep"."EM - 460"."AV460d-1".CW.ENABLE := True;
   MachineConfig[13]."Unit Sep"."EM - 460"."AV460d-1".FB_OPN_ADD := 214;
   MachineConfig[13]."Unit Sep"."EM - 460"."AV460d-1".FB_CLS_ADD := 215;
   MachineConfig[13]."Unit Sep"."EM - 600"."AV615-1".CW.ENABLE := True;
   MachineConfig[13]."Unit Sep"."EM - 600"."FIS615-1".CW.ENABLE := True;
   MachineConfig[13]."Unit Sep"."EM - 600"."FIS615-1".CW.EXIST := True;
   MachineConfig[13]."Unit Sep"."EM - 600"."FIS635-1".CW.ENABLE := True;
   MachineConfig[13]."Unit Sep"."EM - 730".TS730.CW.ENABLE := True;
   MachineConfig[13]."Unit Sep"."EM - 730".TS730.CW.EXIST := True;
   MachineConfig[13]."Unit Sep"."EM - 730".TT730a.CW.ENABLE := True;
   MachineConfig[13]."Unit Sep"."EM - 730".TT730a.CW.EXIST := True;
   MachineConfig[13]."Unit Sep"."EM - 730".TT730a.Address := 128;
   MachineConfig[13]."Unit Sep"."EM - 730".TT731a.Tag := 'TT731a';
   MachineConfig[13]."Unit Sep"."EM - 730".TT731a.CW.ENABLE := True;
   MachineConfig[13]."Unit Sep"."EM - 730".TT731a.CW.EXIST := True;
   MachineConfig[13]."Unit Sep"."EM - 730".TT731a.Address := 130;
   MachineConfig[13]."Unit Sep"."EM - 730".TT731b.CW.ENABLE := True;
   MachineConfig[13]."Unit Sep"."EM - 730".TT731b.CW.EXIST := True;
   MachineConfig[13]."Unit Sep"."EM - 730".TT733.Tag := 'TT733';
   MachineConfig[13]."Unit Sep"."EM - 730".TT733.Address := 132;
   MachineConfig[13]."Unit Sep"."EM - 730".TT734.CW.ENABLE := True;
   MachineConfig[13]."Unit Sep"."EM - 730".TT734.CW.EXIST := True;
   MachineConfig[13]."Unit Sep"."EM - 750".YT75X.CW.ENABLE := TRUE;
   MachineConfig[13]."Unit Process"."EM - 201"."AV201-1".CW.ENABLE := True;
   MachineConfig[13]."Unit Process"."EM - 201"."FIT201-1"."Type" := 2;
   MachineConfig[13]."Unit Process"."EM - 201"."FIT201-1".Address := 256;
   MachineConfig[13]."Unit Process"."EM - 201"."FIT201-1".Max := 100000.0;
   MachineConfig[13]."Unit Process"."EM - 201"."LA201-1".CW.ENABLE := true;
   MachineConfig[13]."Unit Process"."EM - 201"."QT201-1".CW.ENABLE := True;
   MachineConfig[13]."Unit Process"."EM - 201"."QT201-1".CW.EXIST := True;
   MachineConfig[13]."Unit Process"."EM - 201"."QT201-1_OK".CW.ENABLE := True;
   MachineConfig[13]."Unit Process"."EM - 212"."AV212-1".CW.ENABLE := True;
   MachineConfig[13]."Unit Process"."EM - 22X"."AV220-1".CW.ENABLE := True;
   MachineConfig[13]."Unit Process"."EM - 22X"."AV460-1".CW.ENABLE := True;
   MachineConfig[13]."Unit Process"."EM - 22X"."QT220-1".CW.ENABLE := True;
   MachineConfig[13]."Unit Process"."EM - 22X"."PCV22X-1".CW.NO := False;
   MachineConfig[13]."Unit Process"."EM - 22X"."QT220-1_OK".CW.ENABLE := True;
   MachineConfig[13]."Unit Process"."EM - 22X"."QT220-1_OK".CW.EXIST := False;
   MachineConfig[13]."Unit Process"."EM - 22X"."LA220-1".CW.ENABLE := True;
   MachineConfig[13]."Unit Process"."EM - 340"."AV340-1".CW.ENABLE := True;
   MachineConfig[13]."Unit Process"."EM - 340"."AV340-2".CW.ENABLE := True;
   MachineConfig[13]."Unit Process"."EM - 340"."AV460-2".CW.ENABLE := True;
   MachineConfig[13]."Unit Process"."EM - 340"."PIS340-1".CW.ENABLE := True;
   MachineConfig[13]."Unit Dch"."EM - 222"."AV222-1".CW.ENABLE := true;
   MachineConfig[13]."Unit Dch"."EM - 222"."LS222-2".CW.ENABLE := True;
   MachineConfig[13]."Unit Dch"."EM - 222"."LS222-2".CW.EXIST := True;
   MachineConfig[13]."Unit Dch"."EM - 222"."LS222-3".CW.ENABLE := True;
   MachineConfig[13]."Unit Dch"."EM - 222"."LS222-3".CW.EXIST := True;
   MachineConfig[13]."Unit Dch"."EM - 222"."PIT222-1".CW.ENABLE := True;
   MachineConfig[13]."Unit Dch"."EM - 222"."PIT222-1".CW.EXIST := True;
   MachineConfig[13]."Unit Dch"."EM - 222"."TS222-1".CW.ENABLE := True;
   MachineConfig[13]."Unit Dch"."EM - 222"."TS222-1".CW.EXIST := False;
   MachineConfig[13]."Unit Dch"."EM - 222"."TT222-1".CW.ENABLE := True;
   MachineConfig[13]."Unit Dch"."EM - 222"."TT222-1".CW.EXIST := True;
   MachineConfig[13]."Unit Dch"."EM - 300"."AV301-1".CW.ENABLE := True;
   MachineConfig[13]."Unit Dch"."EM - 300"."AV302-1".CW.ENABLE := True;
   MachineConfig[13]."Unit Dch"."EM - 300"."AV303-1".CW.ENABLE := True;
   MachineConfig[13]."Unit Dch"."EM - 300"."AV304-1".CW.ENABLE := True;
   MachineConfig[13]."Unit Dch"."EM - 300"."AV305-1".CW.ENABLE := True;
   MachineConfig[13]."Unit Dch"."EM - 300"."AV306-1".CW.ENABLE := True;
   MachineConfig[13]."Unit Dch"."EM - 300"."AV320-1".CW.ENABLE := True;
   MachineConfig[13]."Unit Dch"."EM - 300"."AV635-1".CW.ENABLE := True;
   MachineConfig[13]."Unit Dch"."EM - 375"."AV37X-1".CW.ENABLE := True;
   MachineConfig[13]."Unit Dch"."EM - 375"."PT37X-1".CW.ENABLE := True;
   MachineConfig[13]."Unit Dch"."EM - 375"."PT37X-1".CW.EXIST := True;
   MachineConfig[13]."Unit Dch"."EM - 506"."AV543-1".CW.ENABLE := true;
   MachineConfig[13]."Unit Dch"."EM - 506".IP506a.CW.ENABLE := True;
   MachineConfig[13]."Unit Dch"."EM - 506".IP506a.CW.EXIST := True;
   MachineConfig[13]."Unit Dch"."EM - 506"."PV376-1".CW.ENABLE := TRUE;
   MachineConfig[13]."Unit Dch"."EM - 506"."PV376-2".CW.ENABLE := TRUE;
   MachineConfig[13]."Unit Dch"."EM - 506".AVDCH.TAG := '506b';
   MachineConfig[13]."Unit Dch"."EM - 506".AVDCH.CW.ENABLE := true;
   MachineConfig[13].Options."EM - 208"."FIT208-1"."Type" := 2;
   MachineConfig[13].Options."EM - 208"."FIT208-1".Address := 266;
   MachineConfig[13].Options."EM - 208"."FIT208-1".Max := 20000.0;
   MachineConfig[13].Communications."EM - BC-COMM".BCI0 := 8;
   MachineConfig[13].Communications."EM - BC-COMM".BCI1 := 8;
   MachineConfig[13].Communications."EM - BC-COMM".BCI2 := 8;
   MachineConfig[13].Communications."EM - BC-COMM".BCI3 := 8;
   MachineConfig[13].Communications."EM - BC-COMM".BCO0 := 8;
   MachineConfig[13].Communications."EM - BC-COMM".BCO1 := 8;
   MachineConfig[13].Communications."EM - BC-COMM".BCO2 := 8;
   MachineConfig[13].Communications."EM - BC-COMM".BCO3 := 8;
   MachineConfig[13].Communications."EM - BC-COMM".ALARM := 8;
   MachineConfig[14].Machine."Family" := 1;
   MachineConfig[14].Machine.TypeNo := 14;
   MachineConfig[14].Machine.Range := 1;
   MachineConfig[14].Machine.SepType := 1;
   MachineConfig[14].Machine.Frame := 2;
   MachineConfig[14].Machine.DchSystem := 3;
   MachineConfig[14].Machine.Spare_1 := 1;
   MachineConfig[14].Machine.FeedPump := 1;
   MachineConfig[14].Machine.Blending := 1;
   MachineConfig[14].Machine.Recirculation := 1;
   MachineConfig[14].Machine.CoolingRecirculation := 1;
   MachineConfig[14].Machine.Spare_2 := 1;
   MachineConfig[14].Machine.eMotion := 1;
   MachineConfig[14].Machine.ConditionAlert := 1;
   MachineConfig[14].Machine.eWON := 1;
   MachineConfig[14].Machine.ALBufferTank := 1;
   MachineConfig[14]."Unit Sep"."EM - 100"."L-GREEN".CW.ENABLE := True;
   MachineConfig[14]."Unit Sep"."EM - 100"."L-GREEN".Address := 162;
   MachineConfig[14]."Unit Sep"."EM - 100"."L-YELLOW".CW.ENABLE := True;
   MachineConfig[14]."Unit Sep"."EM - 100"."L-YELLOW".Address := 163;
   MachineConfig[14]."Unit Sep"."EM - 100"."L-RED".Address := 164;
   MachineConfig[14]."Unit Sep"."EM - 100"."L-BUZZ".Address := 165;
   MachineConfig[14]."Unit Sep"."EM - 100".UPS.CW.EXIST := True;
   MachineConfig[14]."Unit Sep"."EM - 100"."CA VIB WARN".Address := 183;
   MachineConfig[14]."Unit Sep"."EM - 100"."CA VIB ALM".Address := 184;
   MachineConfig[14]."Unit Sep"."EM - 100"."CA ERROR".Address := 191;
   MachineConfig[14]."Unit Sep"."EM - 100"."CA WD".Address := 192;
   MachineConfig[14]."Unit Sep"."EM - 400"."AV409-1".ACT_OUT_ADD := 325;
   MachineConfig[14]."Unit Sep"."EM - 400"."FCV409-1".CW.ENABLE := False;
   MachineConfig[14]."Unit Sep"."EM - 400"."FIS412-1".CW.ENABLE := True;
   MachineConfig[14]."Unit Sep"."EM - 400"."FIS412-1".CW.EXIST := False;
   MachineConfig[14]."Unit Sep"."EM - 400"."FIS412-1".Address := 173;
   MachineConfig[14]."Unit Sep"."EM - 400"."FIT409-1".CW.ENABLE := False;
   MachineConfig[14]."Unit Sep"."EM - 400"."FIT412-1".CW.ENABLE := True;
   MachineConfig[14]."Unit Sep"."EM - 400"."FIT412-1".Address := 78;
   MachineConfig[14]."Unit Sep"."EM - 400"."TT411-1".CW.ENABLE := True;
   MachineConfig[14]."Unit Sep"."EM - 400"."TT411-1".Address := 184;
   MachineConfig[14]."Unit Sep"."EM - 400"."TT41X-1".Tag := 'TT412-1';
   MachineConfig[14]."Unit Sep"."EM - 400"."TT41X-1".CW.ENABLE := True;
   MachineConfig[14]."Unit Sep"."EM - 400"."TT41X-1".CW.EXIST := False;
   MachineConfig[14]."Unit Sep"."EM - 400"."TT41X-1".Address := 190;
   MachineConfig[14]."Unit Sep"."EM - 420".FS421a.CW.ENABLE := True;
   MachineConfig[14]."Unit Sep"."EM - 420".FS421a.Address := 174;
   MachineConfig[14]."Unit Sep"."EM - 420".FS421b.CW.ENABLE := True;
   MachineConfig[14]."Unit Sep"."EM - 420".FS421b.Address := 175;
   MachineConfig[14]."Unit Sep"."EM - 420".LS422a.CW.ENABLE := True;
   MachineConfig[14]."Unit Sep"."EM - 420".LS422a.Address := 176;
   MachineConfig[14]."Unit Sep"."EM - 420"."LS42X(b)".CW.ENABLE := True;
   MachineConfig[14]."Unit Sep"."EM - 420"."LS42X(b)".Address := 177;
   MachineConfig[14]."Unit Sep"."EM - 420"."LS422-1".CW.ENABLE := True;
   MachineConfig[14]."Unit Sep"."EM - 420"."LS422-1".Address := 180;
   MachineConfig[14]."Unit Sep"."EM - 420"."P403-1".CW.ENABLE := True;
   MachineConfig[14]."Unit Sep"."EM - 420"."P421-1".CW.ENABLE := True;
   MachineConfig[14]."Unit Sep"."EM - 420"."P421-1".OUT_ACT_ADD := 336;
   MachineConfig[14]."Unit Sep"."EM - 420"."PV421-1".CW.ENABLE := True;
   MachineConfig[14]."Unit Sep"."EM - 420"."PV421-1".ACT_OUT_ADD := 335;
   MachineConfig[14]."Unit Sep"."EM - 460"."AV460d-1".CW.ENABLE := True;
   MachineConfig[14]."Unit Sep"."EM - 460"."AV460d-1".FB_OPN_ADD := 226;
   MachineConfig[14]."Unit Sep"."EM - 460"."AV460d-1".FB_CLS_ADD := 227;
   MachineConfig[14]."Unit Sep"."EM - 460"."AV460d-1".ACT_OUT_ADD := 193;
   MachineConfig[14]."Unit Sep"."EM - 600"."AV615-1".CW.ENABLE := True;
   MachineConfig[14]."Unit Sep"."EM - 600"."AV615-1".ACT_OUT_ADD := 326;
   MachineConfig[14]."Unit Sep"."EM - 600"."FIS615-1".CW.ENABLE := True;
   MachineConfig[14]."Unit Sep"."EM - 600"."FIS635-1".Tag := 'FIS635a-1';
   MachineConfig[14]."Unit Sep"."EM - 600"."FIS635-1".CW.ENABLE := True;
   MachineConfig[14]."Unit Sep"."EM - 730".TT730a.CW.ENABLE := True;
   MachineConfig[14]."Unit Sep"."EM - 730".TT730a.Address := 176;
   MachineConfig[14]."Unit Sep"."EM - 730".TT730b.CW.ENABLE := True;
   MachineConfig[14]."Unit Sep"."EM - 730".TT730b.Address := 186;
   MachineConfig[14]."Unit Sep"."EM - 730".TT731a.CW.ENABLE := True;
   MachineConfig[14]."Unit Sep"."EM - 730".TT731a.Address := 178;
   MachineConfig[14]."Unit Sep"."EM - 730".TT734.CW.ENABLE := True;
   MachineConfig[14]."Unit Sep"."EM - 730".TT734.Address := 188;
   MachineConfig[14]."Unit Sep"."EM - 750".YT75X.Address := 72;
   MachineConfig[14]."Unit Process"."EM - 201"."AV201-1".FB_OPN_ADD := 201;
   MachineConfig[14]."Unit Process"."EM - 201"."AV201-1".FB_CLS_ADD := 200;
   MachineConfig[14]."Unit Process"."EM - 201"."AV201-1".ACT_OUT_ADD := 180;
   MachineConfig[14]."Unit Process"."EM - 201"."FIT201-1"."Type" := 2;
   MachineConfig[14]."Unit Process"."EM - 201"."FIT201-1".Address := 256;
   MachineConfig[14]."Unit Process"."EM - 201"."FIT201-1".Max := 100000.0;
   MachineConfig[14]."Unit Process"."EM - 201"."LA201-1".Address := 160;
   MachineConfig[14]."Unit Process"."EM - 201"."QT201-1".CW.ENABLE := True;
   MachineConfig[14]."Unit Process"."EM - 201"."QT201-1".CW.EXIST := True;
   MachineConfig[14]."Unit Process"."EM - 201"."QT201-1_OK".CW.ENABLE := True;
   MachineConfig[14]."Unit Process"."EM - 212"."AV212-1".CW.ENABLE := True;
   MachineConfig[14]."Unit Process"."EM - 212"."AV212-1".FB_OPN_ADD := 202;
   MachineConfig[14]."Unit Process"."EM - 212"."AV212-1".FB_CLS_ADD := 203;
   MachineConfig[14]."Unit Process"."EM - 212"."AV212-1".ACT_OUT_ADD := 181;
   MachineConfig[14]."Unit Process"."EM - 22X"."AV220-1".CW.ENABLE := True;
   MachineConfig[14]."Unit Process"."EM - 22X"."AV220-1".FB_OPN_ADD := 205;
   MachineConfig[14]."Unit Process"."EM - 22X"."AV220-1".FB_CLS_ADD := 204;
   MachineConfig[14]."Unit Process"."EM - 22X"."AV220-1".ACT_OUT_ADD := 182;
   MachineConfig[14]."Unit Process"."EM - 22X"."AV460-1".CW.ENABLE := True;
   MachineConfig[14]."Unit Process"."EM - 22X"."AV460-1".FB_OPN_ADD := 222;
   MachineConfig[14]."Unit Process"."EM - 22X"."AV460-1".FB_CLS_ADD := 223;
   MachineConfig[14]."Unit Process"."EM - 22X"."AV460-1".ACT_OUT_ADD := 191;
   MachineConfig[14]."Unit Process"."EM - 22X"."QT220-1".CW.ENABLE := True;
   MachineConfig[14]."Unit Process"."EM - 22X"."QT220-1_OK".CW.ENABLE := true;
   MachineConfig[14]."Unit Process"."EM - 22X"."QT220-1_OK".CW.EXIST := False;
   MachineConfig[14]."Unit Process"."EM - 22X"."LA220-1".CW.ENABLE := True;
   MachineConfig[14]."Unit Process"."EM - 340"."AV340-1".FB_OPN_ADD := 217;
   MachineConfig[14]."Unit Process"."EM - 340"."AV340-1".FB_CLS_ADD := 216;
   MachineConfig[14]."Unit Process"."EM - 340"."AV340-1".ACT_OUT_ADD := 187;
   MachineConfig[14]."Unit Process"."EM - 340"."AV340-2".CW.ENABLE := True;
   MachineConfig[14]."Unit Process"."EM - 340"."AV340-2".FB_OPN_ADD := 221;
   MachineConfig[14]."Unit Process"."EM - 340"."AV340-2".FB_CLS_ADD := 220;
   MachineConfig[14]."Unit Process"."EM - 340"."AV340-2".ACT_OUT_ADD := 190;
   MachineConfig[14]."Unit Process"."EM - 340"."AV460-2".CW.ENABLE := True;
   MachineConfig[14]."Unit Process"."EM - 340"."AV460-2".FB_OPN_ADD := 224;
   MachineConfig[14]."Unit Process"."EM - 340"."AV460-2".FB_CLS_ADD := 225;
   MachineConfig[14]."Unit Process"."EM - 340"."AV460-2".ACT_OUT_ADD := 192;
   MachineConfig[14]."Unit Process"."EM - 340"."PIS340-1".CW.ENABLE := True;
   MachineConfig[14]."Unit Dch"."EM - 222"."AV222-1".CW.ENABLE := True;
   MachineConfig[14]."Unit Dch"."EM - 222"."AV222-1".FB_OPN_ADD := 210;
   MachineConfig[14]."Unit Dch"."EM - 222"."AV222-1".FB_CLS_ADD := 211;
   MachineConfig[14]."Unit Dch"."EM - 222"."AV222-1".ACT_OUT_ADD := 184;
   MachineConfig[14]."Unit Dch"."EM - 222"."LS222-1".Address := 163;
   MachineConfig[14]."Unit Dch"."EM - 222"."TS222-1".CW.EXIST := False;
